# B&R Automation Studio project AriesV2
Automation Studio 4.2.7.54 SP

## Configuration Config_Deployment

### Hardware
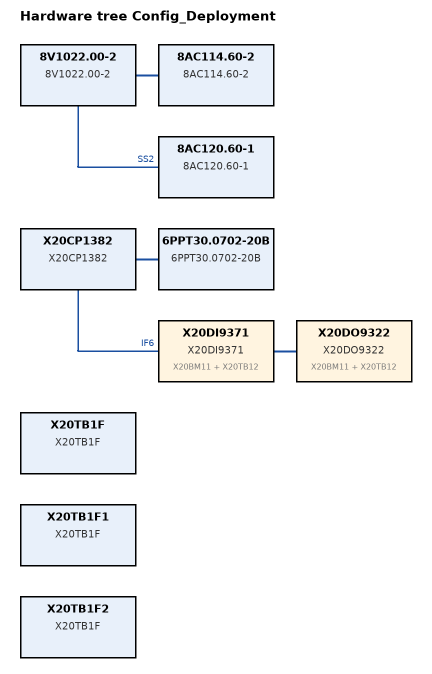
```
6PPT30.0702-20B : 6PPT30.0702-20B v1.1.0.0  [ETH1 -> X20CP1382.IF2 (NodeNumber=1)]
  Terminal = true
  Startmode = 1
  ShowBootlogoVNC = 1
  Mode = Manual
  InternetAddress = 192.168.10.20
  DefaultGateway = 192.168.10.1
  Subnetmask = 255.255.255.0
  Displaybrightness = 75
  SelectedFavoriteVNC = 192.168.10.10
  Favorites_VNC1 = 192.168.10.10
  PasswordVNC = 
  PasswordCIFS = 
  PasswordService = 
  PPTImage = PPT_30_V1.1.1
  VncRefreshRate = 200
8AC114.60-2 : 8AC114.60-2 v1.0.0.8  [SS -> 8V1022.00-2.SS1; PLK1 -> X20CP1382.IF3 (NodeNumber=2)]
8AC120.60-1 : 8AC120.60-1 v1.0.0.2  [SS -> 8V1022.00-2.SS2]
8V1022.00-2 : 8V1022.00-2 v1.0.0.2
  AxisIsPeriodic_r1 = on
  BothEndSwitchesAreNormallyOpen_r1 = on
  QuickStopIsNormallyOpen_r1 = on
X20BM11 : X20BM11 v1.0.0.1  [X2X1 -> X20CP1382.IF6]
X20BM11a : X20BM11 v1.0.0.1  [X2X1 -> X20BM11.X2X2]
X20CP1382 : X20CP1382 v1.3.0.0  [X1 -> X1.SL; X2 -> X2.SL; X3 -> X3.SL]
  Module X1 (Type=X1, Virtual=true, Version=1.0.0.0)
    Connection (Connector=SS1, TargetModule=X20TB1F, TargetConnector=SS)
    Connection (Connector=SL, TargetModule=X20CP1382, TargetConnector=X1)
  Module X2 (Type=X2, Virtual=true, Version=1.0.0.0)
    Connection (Connector=SS1, TargetModule=X20TB1F1, TargetConnector=SS)
    Connection (Connector=SL, TargetModule=X20CP1382, TargetConnector=X2)
  Module X3 (Type=X3, Virtual=true, Version=1.0.0.0)
    Connection (Connector=SS1, TargetModule=X20TB1F2, TargetConnector=SS)
    Connection (Connector=SL, TargetModule=X20CP1382, TargetConnector=X3)
  Connector IF2:
    ActivateDevice = 1
    HostName = x20cpu
    Mode = Manual
    InternetAddress = 192.168.10.10
    SubnetMask = 255.255.255.0
    InaNodeNumber = 0
    Vnc1
    VncVcObjectName1 = Visup
    VncKeyMappingFile1 = VC\PS2-Keyboard4.dis
    VncRefreshRate1 = 200
  Connector IF3:
    CycleTime = 4000
  Connector IF6:
    CycleTime = 4000
  ConfigurationID = AriesV2_Config_Test
  UserPartitionSize = 256
  Simulation = 1
  UserRamSize = 5000
  RemMemSize = 25000
  PermanentPvSize = 15000
  VolatileGlobalPvSize = 300000
  RebootReset = 2
  RebootPowerfail = 2
  TimerDeviceType = EPLX2X
  TimerDevice = X20CP1382.IF3
  TaskClassIdleTime = 8000
  Cyclic1Duration = 4000
  Cyclic1Tolerance = 0
  Cyclic2Duration = 16000
  Cyclic2Tolerance = 16000
  Cyclic3Duration = 48000
  Cyclic3Tolerance = 48000
  Cyclic4Duration = 96000
  Cyclic4Tolerance = 96000
  Cyclic5Duration = 200000
  Cyclic5Tolerance = 200000
  Cyclic6Duration = 496000
  Cyclic6Tolerance = 496000
  Cyclic7Duration = 1000000
  Cyclic7Tolerance = 1000000
  Cyclic8Duration = 8000
  Cyclic8Tolerance = 30000000
  FileDevice1
  FileDeviceName1 = ROOT
  FileDevicePath1 = F:\
  FileDevice2
  FileDeviceName2 = Config
  FileDevicePath2 = F:\Config
  FileDevice3
  FileDeviceName3 = Recipe
  FileDevicePath3 = F:\Recipe
  FileDevice4
  FileDeviceName4 = Process
  FileDevicePath4 = F:\Process
  FtpUser1
  FtpUsername1 = admin
  FtpUserPassword1 = tXcQUdKIsoY/H/jtKSqzHLRzyWbO/eZFb+QmJVs8vuM=
  FtpUserSalt1 = fFlgpUU6
  FTPAccessRight1 = 0
  FTPdevice1 = ALL
  FtpUser2
  FtpUsername2 = user
  FtpUserPassword2 = M/sBBWLbPcMSL0ECBo9+NNWk5QFExAfaSSh+paOlJpQ=
  FtpUserSalt2 = diDYFxUT
  FTPAccessRight2 = 0
  FTPMSpath2 = /
X20DI9371 : X20DI9371 v1.0.1.3  [SS1 -> X20TB12.SS; SL -> X20BM11.SL1]
  Supervision = off
X20DO9322 : X20DO9322 v1.0.3.0  [SS1 -> X20TB12a.SS; SL -> X20BM11a.SL1]
  Supervision = off
X20TB12 : X20TB12 v1.0.0.0
X20TB12a : X20TB12 v1.0.0.0
X20TB1F : X20TB1F v1.0.0.0
X20TB1F1 : X20TB1F v1.0.0.0
X20TB1F2 : X20TB1F v1.0.0.0
```

### Acp10map.ncm - X20CP1382/Motion/Acp10map.ncm
```
NcMapping (NcSwId=Acp10, DisabledNodesAreHidden=False)
  NcObject Axis1 (ModuleId=8V1022.00-2, Type=ncAXIS, Channel=1, AcoposSimulation=Off, InitParameter=Axisi, AcoposParameter=Axisa, AdditionalData=PLCopen_ModPos="1000,1" , Disabled=FALSE, ModuleDisabled=FALSE)
  NcObject 8V1045.00-2_ncV_AXIS1 (ModuleId=8V1022.00-2, Type=ncV_AXIS, Channel=1, Disabled=TRUE, ModuleDisabled=FALSE)
```

### Alarm.mpalarmbasic - X20CP1382/mapp/Alarm.mpalarmbasic
```
Element Alarm_MpLink (Type=mpalarmbasic)
  mapp.Alarm.Factory:
    Reactions:
      Reaction[0]:
        Description = Example: Immediate Stop
  Alarms:
    UserAlarm:
      Alarms:
        Alarm[0]:
          Description = Example: Temperature over Tolerance
          Reaction = 1
```

## Configuration Config_Test

### Hardware
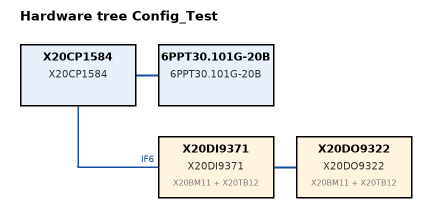
```
6PPT30.101G-20B : 6PPT30.101G-20B v1.1.0.0  [ETH1 -> X20CP1584.IF2 (NodeNumber=1)]
  Terminal = true
  Startmode = 1
  Mode = Manual
  ScreenRotation = 90
  SelectedFavoriteVNC = 192.168.10.10
  PasswordVNC = 
  PasswordCIFS = 
  PasswordService = 
  VncKeyMappingFile = VC\6PPT30.101G-20B.dis
  VncPortNumber = 5901
  VncRefreshRate = 100
  InternetAddress = 192.168.10.20
  DefaultGateway = 192.168.10.1
  Subnetmask = 255.255.255.0
X20BM11 : X20BM11 v1.0.0.1  [X2X1 -> X20CP1584.IF6]
X20BM11a : X20BM11 v1.0.0.1  [X2X1 -> X20BM11.X2X2]
X20CP1584 : X20CP1584 v1.3.2.0
  Connector IF2:
    ActivateDevice = 1
    EthInterfaceRedundant = 0
    HostName = x20cpu
    Mode = Manual
    InternetAddress = 192.168.10.10
    SubnetMask = 255.255.255.0
    Vnc1
    VncVcObjectName1 = Visu1
    VncKeyMappingFile1 = VC\PS2-Keyboard4.dis
    VncRefreshRate1 = 200
  Connector IF3:
    EplInterfaceRedundant = 0
    CycleTime = 8000
    EplEthInterfaceRedundant = 0
  Connector IF6:
    CycleTime = 8000
  ConfigurationID = AriesV2_Config_Test
  UserRamSize = 5000
  RemMemSize = 25000
  PermanentPvSize = 15000
  VolatileGlobalPvSize = 300000
  RebootReset = 2
  RebootPowerfail = 2
  TimerDeviceType = EPLX2X
  TimerDevice = X20CP1584.IF3
  TaskClassIdleTime = 8000
  Cyclic1Duration = 8000
  Cyclic1Tolerance = 0
  Cyclic2Duration = 16000
  Cyclic2Tolerance = 16000
  Cyclic3Duration = 48000
  Cyclic3Tolerance = 48000
  Cyclic4Duration = 96000
  Cyclic4Tolerance = 96000
  Cyclic5Duration = 200000
  Cyclic5Tolerance = 200000
  Cyclic6Duration = 496000
  Cyclic6Tolerance = 496000
  Cyclic7Duration = 1000000
  Cyclic7Tolerance = 1000000
  Cyclic8Duration = 8000
  Cyclic8Tolerance = 30000000
  FileDevice1
  FileDeviceName1 = ROOT
  FileDevicePath1 = F:\
  FileDevice2
  FileDeviceName2 = Config
  FileDevicePath2 = F:\Config
  FileDevice3
  FileDeviceName3 = Recipe
  FileDevicePath3 = F:\Recipe
  FileDevice4
  FileDeviceName4 = Process
  FileDevicePath4 = F:\Process
X20DI9371 : X20DI9371 v1.0.2.0  [SS1 -> X20TB12.SS; SL -> X20BM11.SL1]
  Supervision = off
X20DO9322 : X20DO9322 v1.0.3.0  [SS1 -> X20TB12a.SS; SL -> X20BM11a.SL1]
  Supervision = off
X20TB12 : X20TB12 v1.0.0.0
X20TB12a : X20TB12 v1.0.0.0
```

## Logical view

Binary libraries used (declarations not repeated): operator, runtime, astime, AsIecCon, FileIO, AsXml, standard, brsystem, sys_lib, AsANSL, AsARCfg, AsBrMath, AsBrStr, DataObj, AsTCP, AsUDP, AsUSB, AsArSdm, AsIOTime, AsMem, AsArLog, AsArProf, MTTypes, MTData, wbrListSvc, AsICMP, MpCom, MpAxis, MpWebXs 1.60.1, MpRecipe 1.60.1, MpAlarm, MpFile, Acp10man, Acp10par, NcGlobal, Acp10_MC, Acp10sim, ArTextSys

### BR_AutomationStudio_Winmerge_Settings.txt
```
## This is a directory/file filter for WinMerge
## This filter lets through only files ASP.NET developers care about
name: Exclude Source Control
desc: Exclude Source Control files and directories

## This is an inclusive (loose) filter
## (it lets through everything not specified)
def: include

## Filters for filenames begin with f:
## Filters for directories begin with d:
## (Inline comments begin with " ##" and extend to the end of the line)

## f: \.bzrignore$ ## Bazaar ignore file
## f: \.cvsignore$ ## CVS ignore file
## f: \.gitignore$ ## Git ignore file
## f: \.hgignore$ ## Mercurial ignore file
## f: \.svnignore$ ## Subversion ignore file
## f: \.set$ ## User specific B&R Automation Studio settings
## f: \.state$ ## Even more user specific B&R Automation Studio settings
## f: \.bak$ ## Windows shadow copy files- ignore

f: \.(vs[sp])?scc$  ## Visual SourceSafe files

d: \\\.svn$ ## Subversion working copy
d: \\_svn$  ## Subversion working copy ASP.NET Hack
d: \\cvs$   ## CVS control directory
d: \\\.git$ ## Git directory
d: \\\.bzr$ ## Bazaar branch
d: \\\.hg$ ## Mercurial repository
```

### Global.var
```iecst
VAR CONSTANT
	FORCEIO_ACCESS_LEVEL : UINT := 1;
	CONFIG_ACCESS_LEVEL : UINT := 2;
	RECIPE_ACCESS_LEVEL : UINT := 1;
	DEFINE_MENU_L_HIDE_TIMEOUT_MS : UDINT := 7000;
	DEFINE_MENU_R_HIDE_TIMEOUT_MS : UDINT := 7000;
	DEFINE_HMI_SPLASHSCREEN_TO_MS : UDINT := 5000;
	MAX_IDX_TOTAL_RECIPES : UINT := 100;
	DEFINE_LOGIN_TO : REAL := 600;
END_VAR
(*Insert your comment here.*)
VAR CONSTANT
	MAX_IDX_CREASES : UDINT := 19;
END_VAR
(*Insert your comment here.*)
(*Insert your comment here.*)
VAR RETAIN
	gRecCfg : Global_Par_typ;
END_VAR
VAR
	gAcknowledge : Machine_Alarms_typ;
	gAlarms : Machine_Alarms_typ;
	gMachineName : {REDUND_UNREPLICABLE} STRING[80] := 'Aries';
	gProjectDate : {REDUND_UNREPLICABLE} STRING[80] := '10. April 2017';
	gVersion : {REDUND_UNREPLICABLE} STRING[80] := 'R741';
END_VAR
(*Insert your comment here.*)
VAR
	Axis1 : ACP10AXIS_typ;
	AxisControl : MpAxisBasic;
	AxisPar : MpAxisBasicParType;
	Alarm_Feed : MpAlarmBasicUIConnect20Type := (0);
	Alarm_Feed_UI : MpAlarmBasicUI := (0);
END_VAR
(*Insert your comment here.*)
VAR
	MachineState : AriesMachineState_Enum;
	ProcessState : CreaserPrcsState_Enum;
END_VAR
(*Insert your comment here.*)
VAR
	IO : AriesIOPoints_typ;
	IO_LastCycle : AriesIOPoints_typ;
END_VAR
(*Insert your comment here.*)
VAR
	AppAlarms : MpAlarmBasicUIConnect20Type;
	AppAlarms_FBK : MpAlarmBasic;
	AppAlarms_UI : USINT;
END_VAR
(*Insert your comment here.*)
VAR RETAIN
	gStatistics : Global_Statistics_typ;
END_VAR
(*Insert your comment here.*)
VAR
	gAlarmResetRequested : BOOL;
	StartUIButton_Hide : USINT;
	StopUIButton_Hide : USINT;
	BoardEjectUIButton_Hide : USINT;
	iManualBoardEject : BOOL;
	iMachineErrorReset : BOOL;
	iStartCommand : BOOL;
	iSoftStopCommand : BOOL;
	gSimulateMachine : BOOL;
END_VAR
(*Insert your comment here.*)
VAR CONSTANT
	DEFINE_MM_ROLLER_REV : REAL := 125.664;
END_VAR
VAR
	delta_Board_Position : REAL;
	RollerPos_LastCycle : REAL;
	RollerPos_ThisCycle : REAL;
	Current_Board_Position : REAL;
	Latch_Board_Length : REAL;
	Current_Crease_Section_Length : REAL;
END_VAR
(*Insert your comment here.*)
(*Insert your comment here.*)
```

### Machine.typ
```iecst
TYPE
	CreaserPrcsState_Enum :
		( (*Make sure the indices entered below line up with the VC texts displayed on the UI*)
		PRCS_STATE_INIT := 0,
		PRCS_STATE_READY := 1,
		PRCS_STATE_FEED_BOARD := 2,
		PRCS_STATE_MOVE_CREASE := 3,
		PRCS_STATE_CREASE := 4,
		PRCS_STATE_MOVE_CREASE_WIDTH := 5,
		PRCS_STATE_ERROR := 6,
		PRCS_STATE_EJECT_FINISHED_BOARD := 7,
		PRCS_STATE_SOFT_STOP := 8,
		PRCS_STATE_MOVE_PHOTOEYE_OFFSET := 9
		);
	AriesMachineState_Enum :
		( (*Make sure the indices entered below line up with the VC texts displayed on the UI*)
		MACHINE_STATE_INIT := 0,
		MACHINE_STATE_IDLE := 1,
		MACHINE_STATE_RUNNING := 2,
		MACHINE_STATE_ERROR := 3,
		MACHINE_STATE_HARDWARE_INIT := 4,
		MACHINE_STATE_AXIS_POWER := 5,
		MACHINE_STATE_AXIS_HOME := 6,
		MACHINE_STATE_MANUAL_EJECT := 7
		);
END_TYPE

(*Insert your comment here.*)

TYPE
	CreaserConfig_typ : 	STRUCT
		FeedAxisAccel : REAL;
		FeedAxisDecel : REAL;
		PhotoEyeOffset : REAL;
		PreInsertSpeed : REAL;
		BoardLengthTolerance : REAL;
		CreaseInfeedDelay : REAL;
	END_STRUCT;
	AriesCreaserParams_typ : 	STRUCT
		CreaseDistance_mm : ARRAY[0..MAX_IDX_CREASES]OF REAL;
		CreaseWidth_mm : REAL;
		CreaseCount : UDINT;
		ShaftSensorEdge : UDINT;
		CreaserDirection : UDINT;
		CreaserMotorIdxLag_S : REAL;
		TotalBoardLength : REAL;
	END_STRUCT;
END_TYPE

(*Insert your comment here.*)

TYPE
	AriesIOPoints_typ : 	STRUCT
		oCreaserCCWRotation : BOOL;
		oCreaserCWRotation : BOOL;
		oBoardFeedingLight : BOOL;
		oUIIndicatorLight : BOOL;
		iSafeMachineState : BOOL;
		iCreaserShaftSensor : BOOL;
		iFiberOpticSensor : BOOL;
		iSM1Disabled : BOOL;
	END_STRUCT;
END_TYPE

(*Insert your comment here.*)

TYPE
	Machine_Alarms_typ : 	STRUCT  (*Did something fancy here- structure is copied into array for VC error texts, make sure the following numbers line up with the VC error text indices!*)
		SM1_Disabled : BOOL; (*0*)
		Unsafe_Machine_State : BOOL; (*1*)
		Fiber_Optic_Blocked_RunCmd : BOOL; (*2*)
		Creaser_Shaft_Edge_Timeout : BOOL; (*3*)
		Error_State_Unsafe_Machine : BOOL; (*4*)
		Error_State_SM1_Power : BOOL; (*5*)
		Feed_Axis_Motor_Error : BOOL; (*6*)
		Crease_Count_Greater_Max : BOOL; (*7*)
		Error_State_Process_Error : BOOL; (*8*)
		Load_Recipe : BOOL; (*9*)
		Manual_Home_Creaser_Blade : BOOL; (*10*)
		Board_Length_GT_Confgd_Amount : BOOL; (*11*)
		Board_Length_LT_Confgd_Amount : BOOL; (*12*)
		Measured_Length_GT_Configured : BOOL; (*13*)
		Measured_Length_LT_Configured : BOOL; (*14*)
		Unsaved_Recipe_Params : BOOL; (*15*)
	END_STRUCT;
	Global_Statistics_typ : 	STRUCT
		total_runtime : UDINT;
		runtime_h : UDINT;
		runtime_m : UDINT;
		runtime_s : UDINT;
		total_processed : UDINT;
		Reset : BOOL;
		total_creases : UDINT;
		Sum_Board_Travel_Lengths : REAL;
		Avg_Board_Length : REAL;
	END_STRUCT;
END_TYPE
```

### Generic_Rec_Cfg.typ
```iecst
TYPE
	HMIConfig_typ : 	STRUCT
		passwordSetup : STRING[15];
		passwordEngineer : STRING[15];
		passwordFactory : STRING[15];
		MachineLang : UDINT;
	END_STRUCT;
END_TYPE

(*Insert your comment here.*)

TYPE
	Global_Rec_typ : 	STRUCT
		MagicPrefix : UDINT;
		FeedVelocity : REAL;
		Crease : AriesCreaserParams_typ;
		MagicSuffix : UDINT;
	END_STRUCT;
	Global_Cfg_typ : 	STRUCT
		MagicPrefix : UDINT;
		Creaser : CreaserConfig_typ;
		HMI : HMIConfig_typ;
		wbrMemService : wbrMemService_typ;
		cfgCompile : cfgCompileVersionInfo_typ;
		MagicSuffix : UDINT;
	END_STRUCT;
END_TYPE

(*Insert your comment here.*)

TYPE
	Global_Rec_Cfg_typ : 	STRUCT
		Rec : Global_Rec_typ;
		Cfg : Global_Cfg_typ;
	END_STRUCT;
	Global_RecCfg_Public_In_typ : 	STRUCT
		Copy_default_to_save : USINT;
		Copy_default_to_active : USINT;
		Copy_save_to_active : USINT;
		Copy_save_to_default : USINT;
		Copy_active_to_save : USINT;
		Copy_active_to_default : USINT;
		Copy_internal_to_default : USINT;
		FileName : STRING[255];
	END_STRUCT;
	Global_RecCfg_Public_Out_typ : 	STRUCT
		save_differs_from_active : USINT;
		default_differs_from_save : USINT;
		active_differs_from_default : USINT;
		Initial_Load : USINT;
	END_STRUCT;
	Global_Rec_Cfg_Info_typ : 	STRUCT
		O : Global_RecCfg_Public_Out_typ;
		I : Global_RecCfg_Public_In_typ;
	END_STRUCT;
	Global_Rec_Cfg_IO_typ : 	STRUCT
		Rec : Global_Rec_Cfg_Info_typ;
		Cfg : Global_Rec_Cfg_Info_typ;
	END_STRUCT;
	Global_Par_typ : 	STRUCT
		save : Global_Rec_Cfg_typ;
		active : Global_Rec_Cfg_typ;
		defaultvals : Global_Rec_Cfg_typ;
		IO : Global_Rec_Cfg_IO_typ;
	END_STRUCT;
END_TYPE

(*Insert your comment here.*)
```

### Package Logical/Libraries - Global libraries

### Library Logical/Libraries/jgLibC (ANSIC)
Depends on: standard

#### Indexer_Helper_functions.c
```c
/********************************************************************
 * COPYRIGHT -- Microsoft
 ********************************************************************
 * Library: jgLibC
 * File: Indexer_Helper_functions.c
 * Author: Admin
 * Created: May 11, 2015
 *******************************************************************/

#include <bur/plctypes.h>
#include <jgLibC.h>
UDINT Tms(REAL in){
	UDINT var_return = 0;

	var_return = (UDINT) (1000 * in);

	return var_return;
}
```

### Library Logical/Libraries/MAPPSuppor (ANSIC) - library (written/managed by J. Glisson) containing functions for ACPu err acknowledgement, HMI param table construction, HMI param table activation to the common layer

#### HMIparamList.typ
```iecst
(********************************************************************
 * COPYRIGHT -- piedmont
 ********************************************************************
 * Package: HMI
 * File: HMI.typ
 * Author: goran
 * Created: August 28, 2013
 ********************************************************************
 * Data types of package HMI
 ********************************************************************)
(*########################################################################*)
(*HMI object - PARAMETER LIST - LIMITS*)
(*########################################################################*)
(*########################################################################*)
(*HMI object - PARAMETER LIST*)
(*########################################################################*)

TYPE
	HMITableIndex_enum :
		(
		TABLE_RECIPE := 0,
		TABLE_CONFIG := 1
		);
	hmiTableStatStruct_typ : 	STRUCT
		maxLenDesc : UDINT;
		maxLenName : UDINT;
		Param : UDINT;
		Default : UDINT;
		Min : UDINT;
		Max : UDINT;
		Hide : UDINT;
	END_STRUCT;
	hmiTableStats_typ : 	STRUCT
		Overall : hmiTableStatStruct_typ;
	END_STRUCT;
	PVList_Language_Texts_typ : 	STRUCT
		PVTextLangSpecific : STRING[DEFINE_PAR_NAME_MAXLEN];
		PVDescLangSpecific : STRING[DEFINE_PAR_DESC_MAXLEN];
	END_STRUCT;
	PVListTexts_Info_typ : 	STRUCT
		Str : STRING[DEFINE_PAR_NAME_MAXLEN];
		isValid : BOOL;
		isPV : BOOL;
		isConstant : BOOL;
		Const_Value : REAL;
		PVAdr : {REDUND_UNREPLICABLE} UDINT;
		PVLen : USINT;
		PVDim : USINT;
		PVTyp : UDINT;
		StrLen : UDINT;
	END_STRUCT;
	PVTable_Val_Info_typ : 	STRUCT
		Param : PVListTexts_Info_typ;
		Default : PVListTexts_Info_typ;
		Min : PVListTexts_Info_typ;
		Max : PVListTexts_Info_typ;
		Hide : PVListTexts_Info_typ;
	END_STRUCT;
	PVTableInfo : 	STRUCT
		PVText : ARRAY[0..MAX_IDX_LANGUAGES]OF PVList_Language_Texts_typ;
		Val : PVTable_Val_Info_typ;
		Error : BOOL;
	END_STRUCT;
	HMI_Table_Data_typ : 	STRUCT
		info : ARRAY[0..DEFINE_MAX_TABLE_ENTRIES]OF PVTableInfo;
		Max_Idx_Entries : UDINT;
		Table_Name : STRING[DEFINE_PAR_NAME_MAXLEN];
		NameSpace : STRING[DEFINE_PAR_NAME_MAXLEN];
		Load_OK : BOOL;
	END_STRUCT;
	hmiParamLimits_typ : 	STRUCT
		k_factor : REAL; (*scaling k factor (y=kx + n, where y=dsiplay value, x=plc value)*)
		n_factor : REAL; (*scaling n factor (y=kx + n, where y=dsiplay value, x=plc value)*)
		minValue : REAL; (*min value*)
		maxValue : REAL; (*max value*)
		defaultValue : REAL; (*default value*)
		pEnumText : UDINT; (*ptr to a string of comma delimited enum texts*)
		pEnumVals : UDINT; (*ptr to a string of comma delimited enum values*)
		valueType : UINT; (*type of the paramvalue (0-DINT, 1-REAL, 2-ENUM)*)
	END_STRUCT;
	hmiParamListTable_typ : 	STRUCT
		listHeader : STRING[DEFINE_PAR_NAME_MAXLEN]; (*name of the list (header text)*)
		listIdText : ARRAY[0..DEFINE_MAX_TABLE_ENTRIES]OF STRING[DEFINE_PAR_IDX_MAXLEN]; (*table colum: id-s*)
		listTypeText : ARRAY[0..DEFINE_MAX_TABLE_ENTRIES]OF STRING[DEFINE_PAR_NAME_MAXLEN]; (*table colum: value*)
		listDefaultText : ARRAY[0..DEFINE_MAX_TABLE_ENTRIES]OF STRING[DEFINE_PAR_NAME_MAXLEN]; (*table colum: value*)
		listMinText : ARRAY[0..DEFINE_MAX_TABLE_ENTRIES]OF STRING[DEFINE_PAR_NAME_MAXLEN]; (*table colum: value*)
		listMaxText : ARRAY[0..DEFINE_MAX_TABLE_ENTRIES]OF STRING[DEFINE_PAR_NAME_MAXLEN]; (*table colum: value*)
		listValueText : ARRAY[0..DEFINE_MAX_TABLE_ENTRIES]OF STRING[DEFINE_PAR_NAME_MAXLEN]; (*table colum: value*)
		listName : ARRAY[0..DEFINE_MAX_TABLE_ENTRIES]OF STRING[DEFINE_PAR_NAME_MAXLEN]; (*table colum: name*)
		listDescription : ARRAY[0..DEFINE_MAX_TABLE_ENTRIES]OF STRING[DEFINE_PAR_DESC_MAXLEN]; (*table colum: description*)
		listValuePtr : ARRAY[0..DEFINE_MAX_TABLE_ENTRIES]OF UDINT; (*list of ptrs to parametars*)
		listDecPlaces : ARRAY[0..DEFINE_MAX_TABLE_ENTRIES]OF DINT; (*list of dec places for each parametar*)
		listLimits : ARRAY[0..DEFINE_MAX_TABLE_ENTRIES]OF hmiParamLimits_typ;
		selName : {REDUND_UNREPLICABLE} STRING[DEFINE_PAR_NAME_MAXLEN]; (*name of the currently selected/active parametar*)
		selDescription : STRING[DEFINE_PAR_DESC_MAXLEN]; (*description of the currently selected/active parametar*)
		selValueEnumIndex : UDINT; (*value of the currently selected/active parametar for type enum*)
		selValueEnumIndexMax : UDINT; (*value of the currently selected/active parametar for type enum*)
		selValueREAL : REAL; (*value of the currently selected/active parametar*)
		selValueREALOld : REAL; (*value of the currently selected/active parametar (previous value for change detection*)
		selValueREALMax : REAL; (*max value of the currently selected/active parametar*)
		selValueREALMin : REAL; (*min value of the currently selected/active parametar*)
		selValueREALDefault : REAL; (*default value of the currently selected/active parametar*)
		selValueDecPlaces : DINT; (*default value of the currently selected/active parametar*)
		selValueDINT : DINT; (*value of the currently selected/active parametar*)
		selValueDINTOld : DINT; (*value of the currently selected/active parametar (previous value for change detection*)
		selValueDINTMax : DINT; (*max value of the currently selected/active parametar*)
		selValueDINTMin : DINT; (*min value of the currently selected/active parametar*)
		selValueDINTDefault : DINT; (*default value of the currently selected/active parametar*)
		selValueFormVisible : DINT; (*visibility control of the form / controls for setting parametar value*)
		index : UINT; (*index of the currently selected/active parametar*)
		indexOld : UINT; (*index of the currently selected/active parametar (previous value for change detection)*)
		maxIndex : UINT; (*max index / number of items in the table. Must be less then hmiTableMAXDESCRIPTION!!!*)
		setDefaultRequest : BOOL; (*set default request flag*)
		incDP : USINT;
		decDP : USINT;
	END_STRUCT;
END_TYPE
```

#### hmiParamList.h
```c
/********************************************************************
 * COPYRIGHT -- piedmont
 ********************************************************************
 * Program: hmilogic
 * File: hmiParamList.h
 * Author: goran
 * Created: September 05, 2013
 *******************************************************************/
#include <bur/plctypes.h>
#ifdef _DEFAULT_INCLUDES
#include <AsDefault.h>
#endif
//void hmiParamListTableCyclic(hmiParamListTable_typ* p);
void hmiParamListTableEntryLast(hmiParamListTable_typ* p);
void hmiParamListTableEntryFirst(hmiParamListTable_typ* p, char* pListName);
 void hmiParamListTableAddEntryNext(hmiParamListTable_typ* p, UDINT pValue, char* pName, REAL valDefault, REAL valMin, REAL valMax, DINT decPlaces, REAL k_factor, REAL n_factor, UINT valueType, char* pDescription);
```

#### hmiParamList.c
```c
/********************************************************************
 * COPYRIGHT -- piedmont
 ********************************************************************
 * Program: hmilogic
 * File: hmiParamList.c
 * Author: goran
 * Created: September 05, 2013
 *******************************************************************/

#include <bur/plctypes.h>
#ifdef _DEFAULT_INCLUDES
	#include <AsDefault.h>
#endif

#include <AsBrStr.h>

#define HMI_PARAMLIST_DECPLACES_DEFAULT  2 //default value of decimal places for any real number converted to text. Application specific.

/*
###############################################################################
HMI table editor support. Set of functions that support table based editing of the parametars.
###############################################################################
*/

/**
rouding of a floating point value to the number of required decimal positions.
\param d value
\param pp number of decimal places
\return rounded value

*/
static float roundVal(float d, int ppOffset)
{

	int valInt;
	float exp10topp = 10.0;
	int count = 0;
	int pp = ppOffset;

	if(!pp){
		exp10topp = 1.0;
	}else
		if(pp<0){
		exp10topp = 0.1;
		count = (0 - pp) - 1;
	}else{
		exp10topp = 10.0;
		count = pp - 1;
	}

	while(count--){
		exp10topp *= exp10topp;
	}

	valInt = (int) (d *  exp10topp + 0.5);
	return ( valInt  /  exp10topp  );
}

/**
ftoa (float to ascii converion) with the added support for required number of decimal places in the text ouput.
\param value value to convert
\param pp number of decimal places
\return rounded value

*/
static void ftoaEx(float value, char* pText, int decPlacesOffset)
{
	char text[32];

	int len;
	int comaPos;
	int apendZerosCount;
	int ii;
	float rnd_val;
	int decPlaces = HMI_PARAMLIST_DECPLACES_DEFAULT + decPlacesOffset;

	if(!pText)
		return;

	//limit max dec places
	if(decPlaces > 5)
		decPlaces = 5;

	//convert float to ascii
	//	ftoa(value, text);
	rnd_val = roundVal(value, decPlaces);
	brsftoa(rnd_val , (UDINT)text);

	//get the length of the converted string
	len = strlen(text);
	if(!len){
		//0 length > don't know what to do
		strcpy(pText, "?");
		return;
	}

	//find position of the coma
	comaPos = bgStrFind(text, ".", -1, -1);

	if(!decPlaces){
		//dec places are not needed

		if(comaPos>0){
			//coma is present > terminate the string at the comma position
			text[comaPos] = 0;
		}

	}else{
		//dec places are needed

		if(comaPos<0){
			//no coma present but it is needed
			strcat(text, ".");
			len+=1;
			comaPos=len-1;
		}

		apendZerosCount = decPlaces - (len - comaPos - 1);

		if(apendZerosCount < 0){
			//too many digits after a decimal place > terminate string to a specified number of dec places
			apendZerosCount = 0 - apendZerosCount;
			text[len - apendZerosCount]=0;
		}else{
			//need to add zeros to satisfy the number of dec places
			for(ii=0; ii<apendZerosCount; ii++){
				text[len+ii]='0';
			}
			text[len+ii]=0;
		}
	}

	strcpy(pText, text);
	return;
}

static float hmiParamListTableGetPLCValue(UDINT pValue, REAL k_factor, REAL n_factor, int valueType)
{
	UDINT* pUdint = (UDINT*)pValue;
	float* pFloat = (float*)pValue;
	REAL tempReal;

	switch(valueType){
		case 1:
			if(pFloat){
				tempReal = ((float)(*pFloat)) * k_factor + n_factor;
			}else{
				tempReal = 0.0;
			}
			break;
		default:
			if(pUdint){
				tempReal = ((float)(*pUdint)) * k_factor + n_factor;
			}else{
				tempReal = 0.0;
			}
			break;
	}

	return tempReal;
}

static void hmiParamListTableDisplayToValue(float value, UDINT pValue, char* pOutputText,  int decPlaces, REAL k_factor, REAL n_factor, int valueType)
{
/*
scaling
y=kx + n
y=display value
x=plc value

x = (y- n)*(1/k)

value types:
0-UDINT
1-REAL

*/

	UDINT* pUdint = (UDINT*)pValue;
	float *pFloat = (float*)pValue;

	if(!k_factor){
		strcpy(pOutputText, "ERR: div by 0");
		return;
	}

	switch(valueType){
		case 1:
			*pFloat = (float)((value - n_factor) / k_factor);
			break;
		default:
			*pUdint = (UDINT)((value - n_factor) / k_factor);
			break;
	}

	ftoaEx(value, pOutputText, decPlaces);
}

static void hmiParamListTableValueToDisplay(UDINT pValue, char* pOutputText, float* pOutputFloat, int decPlaces, REAL k_factor, REAL n_factor, int valueType)
{
/*
scaling
y=kx + n
y=display value
x=plc value
*/
	REAL tempReal = hmiParamListTableGetPLCValue(pValue, k_factor, n_factor, valueType);

	if(pOutputFloat)
		*pOutputFloat = tempReal;

	ftoaEx(tempReal, pOutputText, decPlaces);
}

 void hmiParamListTableAddEntryNext(hmiParamListTable_typ* p, UDINT pValue, char* pName,
REAL valDefault, REAL valMin, REAL valMax, DINT decPlaces, REAL k_factor, REAL n_factor, UINT valueType, char* pDescription)
{
	if(p->index >= DEFINE_MAX_TABLE_ENTRIES){
		strcpy(p->listValueText[p->index], "table overflow!");
		return;
	}

	p->listValuePtr[p->index] = pValue;
	bgsprintf(p->listIdText[p->index], "%d", p->index);
	bgStrCpyN(p->listDescription[p->index], pDescription, sizeof(p->listDescription[0]));
	bgStrCpyN(p->listName[p->index], pName, sizeof(p->listName[0]));
	p->listDecPlaces[p->index] = decPlaces;

	switch(valueType){
		case 0:
			bgsprintf(p->listTypeText[p->index], "%s", "INT");
			break;
		case 1:
			bgsprintf(p->listTypeText[p->index], "%s", "FLOAT");
			break;
		default:
			bgsprintf(p->listTypeText[p->index], "%s", "ERR");
			break;
	}

	brsftoa(valDefault,(UDINT) &p->listDefaultText[p->index]);
	brsftoa(valMin,(UDINT) &p->listMinText[p->index]);
	brsftoa(valMax,(UDINT) &p->listMaxText[p->index]);

	p->listLimits[p->index].defaultValue = valDefault;
	p->listLimits[p->index].minValue= valMin;
	p->listLimits[p->index].maxValue= valMax;
	p->listLimits[p->index].k_factor= k_factor;
	p->listLimits[p->index].n_factor= n_factor;
	p->listLimits[p->index].valueType= valueType;

	hmiParamListTableValueToDisplay(p->listValuePtr[p->index],
		p->listValueText[p->index], 0, p->listDecPlaces[p->index], p->listLimits[p->index].k_factor, p->listLimits[p->index].n_factor, p->listLimits[p->index].valueType);

	p->index++;
	p->maxIndex++;
}

void hmiParamListTableEntryFirst(hmiParamListTable_typ* p, char* pListName)
{
	brsmemset((UDINT) p, 0, sizeof(hmiParamListTable_typ));
	p->maxIndex = 0;
	p->index = 0;
	bgStrCpyN(p->listHeader, pListName, sizeof(p->listHeader));
}

void hmiParamListTableEntryLast(hmiParamListTable_typ* p)
{
	if(p->maxIndex)
		p->maxIndex--;

	//init index value
	p->index = 0;

	//update text fields according to the currently selected table element
	bgStrCpyN(p->selName, p->listName[p->index], sizeof(p->selName));
	bgStrCpyN(p->selDescription, p->listDescription[p->index], sizeof(p->selDescription));

	//set limits on the HMI input control that coresponds to the currently selected table element
	p->selValueREALMin = p->listLimits[p->index].minValue;
	p->selValueREALMax= p->listLimits[p->index].maxValue;
	p->selValueREALDefault = p->listLimits[p->index].defaultValue;
	p->selValueDecPlaces = p->listDecPlaces[p->index];

	//display selected table element
	hmiParamListTableValueToDisplay(p->listValuePtr[p->index],
		p->listValueText[p->index], &p->selValueREAL, p->listDecPlaces[p->index], p->listLimits[p->index].k_factor, p->listLimits[p->index].n_factor, p->listLimits[p->index].valueType);

}

USINT hmiParamListTableCyclic(UDINT p_int)
{
	hmiParamListTable_typ* p = p_int;

	//limit index to max index value (up arrow)
	if(p->index >= p->maxIndex){
		p->index = p->maxIndex;
	}

	//keep checking if index changes (i.e. user changes entry selection)
	if(p->index != p->indexOld){
		//index change > update selected value for user entry
		p->indexOld = p->index;
		hmiParamListTableValueToDisplay(p->listValuePtr[p->index], p->listValueText[p->index],
			&p->selValueREAL, p->listDecPlaces[p->index], p->listLimits[p->index].k_factor, p->listLimits[p->index].n_factor, p->listLimits[p->index].valueType);
		//store value for change detection
		p->selValueREALOld = p->selValueREAL;

		//update text fields
		bgStrCpyN(p->selName, p->listName[p->index], sizeof(p->selName));
		bgStrCpyN(p->selDescription, p->listDescription[p->index], sizeof(p->selDescription));

		//set limits for the selected element
		p->selValueREALMin = p->listLimits[p->index].minValue;
		p->selValueREALMax= p->listLimits[p->index].maxValue;
		p->selValueREALDefault = p->listLimits[p->index].defaultValue;
		p->selValueDecPlaces = p->listDecPlaces[p->index];

	}

	//keep checking if currently selected value changes(i.e. user enteres new value)
	if(p->selValueREALOld != p->selValueREAL){
		if(p->selValueREALMin < p->selValueREALMax){
			//enforce limits
			if(p->selValueREAL < p->selValueREALMin)
				p->selValueREAL = p->selValueREALMin;

			if(p->selValueREAL > p->selValueREALMax)
				p->selValueREAL = p->selValueREALMax;
		}
		p->selValueREALOld = p->selValueREAL;
		hmiParamListTableDisplayToValue(p->selValueREAL, p->listValuePtr[p->index], p->listValueText[p->index],
			p->listDecPlaces[p->index], p->listLimits[p->index].k_factor, p->listLimits[p->index].n_factor, p->listLimits[p->index].valueType);
	}

	//keep checking if the source of the currently selected value changes on a PLC(i.e. PLC location gets updated, etc)
	{
		float tempVal = hmiParamListTableGetPLCValue(p->listValuePtr[p->index], p->listLimits[p->index].k_factor, p->listLimits[p->index].n_factor, p->listLimits[p->index].valueType);
		if(p->selValueREAL != tempVal){
			//PLC value changed > update displayed value
			p->selValueREAL = tempVal;
			p->selValueREALOld = p->selValueREAL;
			hmiParamListTableDisplayToValue(p->selValueREAL, p->listValuePtr[p->index], p->listValueText[p->index],
				p->listDecPlaces[p->index], p->listLimits[p->index].k_factor, p->listLimits[p->index].n_factor, p->listLimits[p->index].valueType);

		}
	}

	//set default value request?
	if(p->setDefaultRequest){
		p->setDefaultRequest = 0;
		p->selValueREAL = p->selValueREALDefault;
	}
	return 0;
}

//eof
```

### Package Logical/Libraries/wbrServices - Service libraries

### wbrServices.typ
```iecst
(*** /*****************************************************************
 * \copyright -- Piedmont Automation
 ********************************************************************
 * Program : wbrServices
 * \file :   wbrServices.typ
 * \author : Blanton Radford
 * \date Created: July 17, 2015
 ********************************************************************
 * Data types of package wbrServices
 ***************************************************************/ *****)

TYPE
	wbrSvcBool_enum :
		(
		NO := 0,
		YES,
		OFF := 0,
		ON,
		STOP := 0,
		START,
		UNCHECK := 0,
		CHECK
		);
	cfgFileInfo_typ : 	STRUCT
		timestamp : STRING[63];
		path : STRING[127];
		machineNumber : UDINT;
		machineName : STRING[31];
	END_STRUCT;
END_TYPE
```

### wbrServicesGlobal.var
```iecst
(********************************************************************
 * COPYRIGHT -- Piedmont Automation
 ********************************************************************
 * Package: listServices
 * File: listServicesGlobal.var
 * Author: Blanton Radford
 * Created: August 11, 2014
 ********************************************************************
 * Variables of package listServices
 ********************************************************************)
VAR
	memService : wbrMemService_typ := (0);
	logService : wbrLogService_typ := (0);
	genericPing : wbrPingService_typ;
END_VAR
```

### Program Logical/Libraries/wbrServices/bglibasWBR

#### bgfifo.c
```c
/********************************************************************
 * COPYRIGHT -- HP
 ********************************************************************
 * Library: bglibas
 * File: bgfifo.c
 * Author: goran
 * Created: February 01, 2013
 *******************************************************************/

#include <bur/plctypes.h>
#ifdef __cplusplus
	extern "C"
	{
#endif

#include "bglibasWBR.h"

#ifdef __cplusplus
	};
#endif
#include <string.h>

static void bgFIFOPushEntry(bgFIFO_typ* p)
{
	char *pSrc = (char*)p->iPtrPushData;//src data
	char* pDst = (char*)((char*)p->prvFIFOMemory + (p->cfgEntrySize * p->oPushIdx));//empty FIFO location
	memcpy(pDst, pSrc, p->cfgEntrySize);

	p->oPushIdx++;//inc location index to next empty FIFO spot
	if(p->oPushIdx >= p->cfgMaxEntries){
		p->oPushIdx = 0;//handle roll over (ring buffer)
	}

	p->oFIFOCount++;//inc number of FIFO entries
	if(p->oFIFOCount >= p->cfgMaxEntries){
		p->oFIFOFull = 1;//set FIFO full indication
	}
}

static void bgFIFOPullEntry(bgFIFO_typ* p)
{
	char* pSrc = (char*)((char*)p->prvFIFOMemory + (p->cfgEntrySize * p->oPullIdx));//oldest FIFO entry
	char *pDst = (char*)p->oPtrPullData;//destination
	memcpy(pDst, pSrc, p->cfgEntrySize);

	p->oPullIdx++;//inc oldest stored FIFO entry position
	if(p->oPullIdx >= p->cfgMaxEntries){
		p->oPullIdx = 0;//handle roll over (ring buffer)
	}

	if(p->oFIFOCount)//dec number of entris in the FIFO
		p->oFIFOCount--;

	p->oFIFOFull = 0;//reset FIFO full indication
}

/**
bgFIFOInit()
-simple FIFO. Stores upto (entryTotalCount) number of elements. Elements MUST be of the same size.
-supports push/pull action
-push:
- user supplied data is copied into the available FIFO memory space, number of items in the FIFO gets incremented,
index variable that keeps track of next empty FIFO location is adjusted; if FIFO full - no action, error returned
-pull:
- oldest entry from FIFO copied to user supplied data space; number of items in the FIFO gets decremented,
index variable that keeps track of oldeset FIFO entry is adjusted; if FIFO empty - no action, error is returned
*/
unsigned long bgFIFOInit(struct bgFIFO_typ* p, unsigned long  entrySize, unsigned long  entryTotalCount, unsigned long  pFIFOMem)
{
	if(!p || !pFIFOMem || !entrySize || (entryTotalCount <=5))
		return 1;

	p->iPtrPushData = 0;
	p->oPtrPullData = 0;

	p->oFIFOCount = 0;
	p->oFIFOFull = 0;

	p->cfgEntrySize = entrySize;
	p->cfgMaxEntries = entryTotalCount;
	p->prvFIFOMemory = pFIFOMem;
	p->oPullIdx = 0;
	p->oPushIdx = 0;
	return 0;
}

/* Push data to FIFO. Content from pSrc is copied into the available FIFO memory. In case of error return value is != 0*/
unsigned long bgFIFOPush(struct bgFIFO_typ* p, unsigned long pSrc, unsigned long srcSize)
{
	if(!p)
		return 1;

	if(!p->prvFIFOMemory)
		return 2;

	if(!pSrc)
		return 3;

	if(!srcSize || (srcSize != p->cfgEntrySize) )
		return 4;

	if(p->oFIFOFull)
		return 5;

	p->iPtrPushData = pSrc;
	bgFIFOPushEntry(p);
	return 0;
}

/* Pull (retrive) data from FIFO. Oldest entry from FIFO memory is copied into the provided pDst space. In case of error return value is != 0*/
unsigned long bgFIFOPull(struct bgFIFO_typ* p, unsigned long pDst, unsigned long dstSize)
{
	if(!p)
		return 1;

	if(!p->prvFIFOMemory)
		return 2;

	if(!pDst)
		return 3;

	if(!dstSize || (dstSize != p->cfgEntrySize) )
		return 4;

	if(!p->oFIFOCount)
		return 5;

	p->oPtrPullData = pDst;
	bgFIFOPullEntry(p);
	return 0;
}

/* Get the number of entries stored in the FIFO.*/
unsigned long bgFIFOGetCount(struct bgFIFO_typ* p)
{
	if(!p)
		return 0;

	return p->oFIFOCount;
}

/* Check if FIFO is full.*/
unsigned long bgFIFOIsFull(struct bgFIFO_typ* p)
{
	if(!p)
		return 0;

	return p->oFIFOFull;
}
//EOF
```

#### bgTimer1ms.c
```c
/********************************************************************
 * COPYRIGHT -- belgor
 ********************************************************************
 * Package: bglib
 * File: bgTimer1ms.c
 * Author: goran
 * Created: October 05, 2011
 *******************************************************************/
#include <bur/plctypes.h>
#ifdef __cplusplus
	extern "C"
	{
#endif

#include "bglibasWBR.h"

#ifdef __cplusplus
	};
#endif
#include <standard.h>

/* Timer cyclic function. Must be called cyclicly for corret timer operation. */
unsigned long  bgTimerCyclic(struct TON *timer){
	TON(timer);
	return 0;
}

unsigned long  bgTimerOffCyclic(struct TOF *timer){
	TOF(timer);
	return 0;
}

/* Start timer for a defined amount of time [ms]. IMPORTANT: function uses TON library call. Same restrictions apply! */
unsigned long  bgTimerStart(struct TON *timer, unsigned long timeoutTime){
	timer->IN = 0;
	TON(timer);
	timer->IN = 1;
	timer->PT = timeoutTime;
	TON(timer );
	return 0;
}

/* Stop the timer.*/
unsigned long  bgTimerStop(struct TON *timer){
	timer->IN = 0;
	TON(timer);
	return 0;
}

/* Check if timer has expired.*/
BOOL  bgTimerIsTimeOut(struct TON *timer){
	if( bgTimerIsEnabled(timer) ){
		return (timer->Q);
	}else{
		return (1);
	}
}

/* Check if timer is enabled.*/
BOOL  bgTimerIsEnabled(struct TON *timer){
	return (timer->IN);
}

/* Retrive the remainig timer time [ms].*/
unsigned long  bgTimerTimeRemaining(struct TON *timer){
	return (timer->PT - timer->ET);
}

/* Retrive the elapsed timer time [ms].*/
unsigned long  bgTimerTimeElapsed(struct TON *timer) {
	return (timer->ET);
}

//EOF
```

### Program Logical/Libraries/wbrServices/Cyclic/wbrService

#### wbrServiceCyclic.c
```c
/********************************************************************
 * \copyright -- Piedmont Automation
 ********************************************************************
 * Program : wbrService
 * \file :   wbrServiceCyclic.c
 * \author : Blanton Radford
 * \date Created: May 18, 2015
 ********************************************************************
 * \brief Implementation of program wbrService
 ********************************************************************/

#ifdef _DEFAULT_INCLUDES
  #include <AsDefault.h>
#endif

/*! \brief Cyclic task for ?
*   \pre   Place in TC#?
*/
void _CYCLIC wbrServiceCyclic(void)
{
  //! \todo   check available mem and set flags to increase partition size if needed
  memService.status.blockFree=  memSvcGetMemInfo();

  if(logService.busy)  writeMessagesToLog();

  wbrPingStation(&genericPing);
}

void _EXIT wbrServiceExit(void)
{
  if(logService.busy)  writeMessagesToLog();
}
```

### changeLog.txt
```
0.10.7  2016-04
  Clean up some /todos and other comments
  Added wbrMemService to wrap AsMem and allow services besides list service
    to use heap memory
    moved mem funcs and data from wbrListService to wbrMemService

0.10.6  2016-03-31
  Added TimerServices
    Made a few mods to suit Hailo project and be more generic, e.g. msTimer object declared
    Using clock_ms() from AsTime to count milliseconds
    Added msTimer.diff_ms to facilitate time tracking, e.g. "hour meters"
  A few changes to Init and Cyclic to be more generic for multiple projects
    Write compile info to log on Init
  Updated package dependencies to facilitate more trouble-free importing

0.10.5  2015-10-??
  Initial release
    Used in APDW project
    No complaints as of 2016-03-07
```

### TimerServices.var - Package variables
```iecst
(********************************************************************
 * COPYRIGHT -- Piedmont Automation
 ********************************************************************
 * Package: TimerServices
 * File: TimerServices.var
 * Author: Blanton Radford
 * Created: December 05, 2014
 ********************************************************************
 * Variables of package TimerServices
 ********************************************************************)
VAR
	msTimer : msTimer_typ;
END_VAR
```

- Program Logical/Libraries/wbrServices/TimerServices/msTimeSvc (ANSIC) - ms-based time service (no source held here)

### wbrLogSvc.typ
```iecst
(*** /*****************************************************************
 * \copyright -- Piedmont Automation
 ********************************************************************
 * Program : wbrLogSvc
 * \file :   wbrLogSvc.typ
 * \author : Blanton Radford
 * \date Created: May 07, 2015
 ********************************************************************
 * Data types of library wbrLogSvc
 ****************************************************************/ ****)

TYPE
	wbrLogServiceTextLog_typ : 	STRUCT
		view : ARRAY[0..127]OF STRING[127]; (*View window into the log*)
		str : wbrListSvcStringList_typ;
	END_STRUCT;
	wbrLogServiceLogListNode_typ : 	STRUCT
		fb : AsArLogWrite;
		inMsg : STRING[127];
	END_STRUCT;
	wbrLogService_typ : 	STRUCT
		list : linkedList_typ;
		message : STRING[127] := 'no message to output';
		log : wbrLogServiceTextLog_typ;
		logLevel : USINT := 4; (*The higher the value, the more messages are logged, i.e. the log will contain more detail and will grow larger more quickly*)
		busy : BOOL;
		maxNodesUsed : UDINT;
	END_STRUCT;
	wbrLogServiceLogbookInfo_typ : 	STRUCT
		name : STRING[15];
		length : UDINT := 65535;
		memType : UDINT := 2;
		status : UINT;
		ident : UDINT;
		index : UDINT;
		formatVer : UDINT;
		fb : REFERENCE TO AsArLogGetInfo;
	END_STRUCT;
END_TYPE
```

### Library Logical/Libraries/wbrServices/wbrMemSvc (ANSIC)
Depends on: AsMem

#### wbrMemSvc.typ - Exported data types
```iecst
(*** /*****************************************************************
 * \copyright -- Piedmont Automation
 ********************************************************************
 * Program : wbrMemSvc
 * \file :   wbrMemSvc.typ
 * \author : Blanton Radford
 * \date Created: April 14, 2016
 ********************************************************************
 * Data types of library wbrMemSvc
 ****************************************************************/ ****)

TYPE
	wbrMemSvcStatus_typ : 	STRUCT
		memInitValid : BOOL;
		blockFree : UDINT; (*Size of the largest available heap memory bock*)
	END_STRUCT;
	wbrMemSvcStoredConfig_typ : 	STRUCT
		memRequestSize : UDINT; (*Size of the heap memory partition to be requested during initialization*)
	END_STRUCT;
	wbrMemService_typ : {REDUND_UNREPLICABLE} 	STRUCT
		status : {REDUND_UNREPLICABLE} wbrMemSvcStatus_typ;
		config : REFERENCE TO wbrMemSvcStoredConfig_typ;
	END_STRUCT;
END_TYPE
```

### Library Logical/Libraries/wbrServices/wbrPingSvc (ANSIC)
Depends on: AsICMP, wbrLogSvc, bglibasWBR, AsTime

### bglibasWBR_C.h
```c
/********************************************************************
 * \copyright -- Piedmont Automation
 ********************************************************************
 * Program : wbrServices_C_Includes
 * \file :   bglibasWBR_C.h
 * \author : Blanton Radford
 * \date Created: August 17, 2015
 *******************************************************************/

#include <stdarg.h>

#include <bur/plctypes.h>

UDINT  bgSSMPrintToTextLog(struct bgSSM_typ* p, const char* format, ...);
```

### Library Logical/Libraries/wbrServices/wbrsprintf (ANSIC) - Writes user-formatted output to a string

#### ofmt.c
```c
/*
 *  __ofmt - in-memory text conversion and formatting
 *
 *  __ofmt is used by printf(), fprintf() and sprintf() to format
 *  a string.
 *
 *  A format argument is a string to be output with optional embedded
 *  conversion specifications.  The conversion specifications start with
 *  a `%' and end with a conversion character
 */

#include <stdarg.h>
#include <stdio.h>
#include <limits.h>
#include <ctype.h>
#include <string.h>
/*#include <introl.h>*/
#define FLOATS  /*!!!*/
#define LONGS /*!!!*/

extern void __cvtflasc(double arg, int ndigits, int *decpt, int *sign, char eflag, int bufsize, char *buf);

/* to save space on smaller processors, we will undef
 * all ctype macros, this will cause their functions to be used.
 */
#if defined __CC01__ || defined __CC03__ || defined __CC11__ || defined __CC09__
#undef isalnum
#undef isalpha
#undef iscntrl
#undef isdigit
#undef isgraph
#undef islower
#undef isprint
#undef ispunct
#undef isspace
#undef isupper
#undef isxdigit
#undef __tolower
#undef __toupper
#endif /* use less memory */

/*  LONGINTS will be defined if longs and ints are the same size
 *  on the target.
 */

#if INT_MAX == LONG_MAX
#define LONGINTS 1
#undef LONGS
#else
#define LONGINTS 0
#endif

/*
 * a few typedefs and defines
 */
#ifdef UCHAR
#undef UCHAR
#endif
typedef unsigned char UCHAR;
#ifdef UINT
#undef UINT
#endif
typedef unsigned int UINT;
#ifdef ULONG
#undef ULONG
#endif
typedef unsigned long ULONG;
#ifdef ULLONG                                                                   //  WBR: added 2013-08-21  for future long long support
#undef ULLONG
#endif
typedef unsigned long long ULLONG;                                              //  WBR: added 2013-08-21  for future long long support

#define INITPREC  6 /* number + (opt sign) */
#define MAXLEN 21

static void putcurrent(FILE *stream, char **line, /*int buf_size,*/ int putvalue, int *numberput);

/*
 * definitions for __ofmt flags.
 */
#define INTPAD    0x01
#define LEFTJUST  0x02  /* left justify output */
#define ALTERNATE 0x04  /* use "#" alternate form */
#define LONGFLAG  0x08  /* is this a long argument */
#define SIGNFLAG  0x10  /* must we output a sign */
#define LEADINGZERO 0x20  /* output a leasing zero */
#define PRECISIONFLAG 0x40  /* user specified precision */

#define FLOATFLAG 0x01  /* are we in a float format */
#define DECIMALPOINT  0x02  /* should we output a decimalpoint */
#define EXPSIGN   0x04  /* sign of exponent 0:+, 1:- */
#define EXPONENT  0x08  /* exponent: yes or no */
#define ETYPE   0x10  /* "e" format conversion in __cvtflasc */

int bf_sz;

int __ofmt(FILE *stream, char *line, int buf_size, const char *format, va_list ap)      // WBR: added buf_size
  {
  UCHAR flags;    /* flag holder for output formatting */
  UCHAR fflags;   /* flags for float formatting */
  char  work[MAXLEN]; /* Maximum character length or any float, int, etc. */
  char  *workptr; /* temp pointer used to move through work[] */
  char  c;    /* current character in format string */
  char  base;   /* base for numerical conversions */
  char  sign;   /* (+,-, ,\0) used when SIGNFLAG is set */
  int width;    /* %3: format width: default 0 */
  int precision;  /* %.3: format precision: default -1 */
  int numberput = 0;  /* number of characters output */
  char  pad;    /* character to pad fields with */
  int totallength;  /* Number of spaces to pad determined in each case */
  int numchars; /* number of characters in 'number' */
#ifdef  LONGS
  long  ltemp;    /* long temporary */
  ULONG conv_val; /* variable used by 'convert:' which contains the number */
#else
  int ltemp;    /* int temporary */
  UINT  conv_val; /* variable used by 'convert:' which contains the number */
#endif
  long long lltemp;   // long long temporary                                    WBR: added 2013-08-21  for future long long support
  ULLONG    conv_llval;
  int decpt = 0;  /* double decimal point (needed anyway) */
#ifdef  FLOATS
  int exponent; /* represents the exponent value */
  double  ftemp;    /* double temporary */
  int exponent_begin; /* beginning index into "work[]" for the exponent */
#endif

bf_sz=  buf_size;     // WBR: set buffer size for wbrsnprintf

  while ((c = *format)) /* get a format character */
    {
    if (c != '%') /* if no conversion specifier ... */
      {
      /* just send character */
      putcurrent(stream, &line, c, &numberput);
      ++format;
      continue; /* and try again */
      }

    workptr = work;   /* set up work buffer ptr */
    fflags = flags = 0; /* initial all flag bits to 0 */
    precision = -1;
    width = 0;
    pad = ' ';    /* default padding character */

incloop:  ++format;
loop:   switch (c = *format)
      {
      case ' ':
        flags |= SIGNFLAG;
        sign = ' ';
        goto incloop;
      case '#':
        flags |= ALTERNATE;
        goto incloop;
      case '-':
        flags |= LEFTJUST;
        goto incloop;
      case '+':
        flags |= SIGNFLAG;
        sign = '+';
        goto incloop;
      case '%':
        putcurrent(stream, &line, '%', &numberput);
        ++format;
        break;
      case '0':
        /* set pad character to zero */
        pad = '0';
        goto incloop;
#if defined(LONGS) || defined(LONGINTS)
      case 'l':
        flags |= LONGFLAG;
        goto incloop;
#endif /* LONGFLAGS */
      case '*':
        /* get width */
        width = (va_arg(ap, int));
        if (*(++format) != '.')
          goto loop;
        ++format;
        if (isdigit(*format))
          goto numprecision;
        if (*format != '*')
          goto loop;
argprecision:
        flags |= PRECISIONFLAG;
        precision = va_arg(ap, int);
        goto incloop;
      case '1': case '2': case '3':
      case '4': case '5': case '6':
      case '7': case '8': case '9':
        while(isdigit(*format))
          width = 10 * width + (*(format)++ - '0');
        if (*format == '.')
          {
      case '.':
          /* get the maximum width allowed
           */
          flags |= PRECISIONFLAG;
          precision = 0;
          ++format; /* skip the '.' */

          if (*format == '*')
            goto argprecision;
          else
numprecision:
            while (isdigit(*format))
              precision = 10 * precision +
              (*(format)++ - '0');
          }
        goto loop;
#ifdef  FLOATS
      {
      int negative;

      case 'G':
      case 'g':
        ftemp = (va_arg(ap,double));
        __cvtflasc(ftemp, precision, &decpt, &negative,
          0, sizeof(work), workptr);
        if (decpt < -4 && decpt < precision)
          goto float_common;
        goto set_e_flags;
      case 'E':
      case 'e':
        /* set the E format flag and other float flags */
        ftemp = (va_arg(ap,double));
      set_e_flags:
        fflags |= EXPONENT | ETYPE;
        goto float_common;
      case 'F':
      case 'f':
        ftemp = (va_arg(ap,double));
      float_common:
        fflags |= FLOATFLAG;
        exponent = 0;
        workptr = work;

        if (precision == -1)
          precision = INITPREC;

        __cvtflasc(ftemp, precision, &decpt, &negative,
          fflags & ETYPE, sizeof(work), workptr);

        if (precision != 0)
          fflags |= DECIMALPOINT;

        if (negative)
          {
          flags |= SIGNFLAG;
          sign = '-';
          }

        if (decpt < 0)
          flags |= LEADINGZERO;
        else
          flags &= ~LEADINGZERO;

        if (fflags & EXPONENT)
          {
          if (decpt < 0)
            {
            fflags |= EXPSIGN;
            decpt = -decpt;
            exponent = decpt + 1;
            }
          else
            {
            exponent = decpt - 1;
            fflags &= ~EXPSIGN;
            }
          decpt = 1;
          workptr[MAXLEN-1] = '\0';
          if (exponent > -10 && exponent < 10)
            {
            workptr[MAXLEN-2] = exponent + '0';
            workptr[MAXLEN-3] = '0';
            exponent = 4;
            exponent_begin = MAXLEN - 3;
            }
          else if (exponent > -100 && exponent < 100)
            {
            workptr[MAXLEN-2] = exponent % 10 + '0';
            workptr[MAXLEN-3] = (exponent / 10) % 10 + '0';
            exponent = 4;
            exponent_begin = MAXLEN - 3;
            }
          else
            {
            char *s = workptr + MAXLEN - 1;
            int tmp;
            for (tmp = 0 ; tmp < 3 ; ++tmp)
              {
              *--s = exponent % 10 + '0';
              exponent /= 10;
              }
            exponent = 5;
            exponent_begin = MAXLEN - 4;
            }
          }

        if (decpt > 0)
          totallength = decpt;
        else
          totallength = 1;

        totallength += precision + totallength +
          ((fflags & DECIMALPOINT) != 0) + ((flags & SIGNFLAG) != 0);

        goto output;  /* output */
      }
#endif
      case 'N':
      case 'n':
        *(va_arg(ap, int *)) = numberput;
        continue;
      case 'I':
      case 'i':
      case 'D':
      case 'd':
        /* convert signed `int' or `long' to decimal
         */
#ifdef  LONGS
        if (flags & LONGFLAG)
          {
          ltemp = (va_arg(ap, long));
          if (ltemp < 0)
            {
            flags |= SIGNFLAG;
            ltemp = -ltemp;
            sign = '-';
            }
          }
        else
#endif
          {
          ltemp = (va_arg(ap, int));
          if (ltemp < 0)
            {
            flags |= SIGNFLAG;
            sign = '-';
            ltemp = -ltemp;
            }
          }

        conv_val = ltemp;
        base = 10;
        goto convert;

      case 'U':
      case 'u':
        /* convert unsigned instead of signed
         */
#ifdef  LONGS
        if (flags & LONGFLAG)
          conv_val = (va_arg(ap,unsigned long));
        else
#endif
          conv_val = (va_arg(ap,unsigned));

        /* clear signflag
         */
        flags &= ~SIGNFLAG;
        base = 10;
        goto convert;

      case 'P':
      case 'p':
      case 'X':
      case 'x':
        /* convert to hexadecimal instead of decimal
         */
#ifdef  LONGS
        if (flags & LONGFLAG)
          conv_val = (va_arg(ap,unsigned long));
        else
#endif
          conv_val = (va_arg(ap,unsigned));
        base = 16;
        flags &= ~SIGNFLAG;
        goto convert;

      case 'O':
      case 'o':
        /* convert to octal instead of decimal
         */
#ifdef  LONGS
        if (flags & LONGFLAG)
          conv_val = (va_arg(ap,unsigned long));
        else
#endif
          conv_val = (va_arg(ap,unsigned));

        base = 8;
        flags &= ~SIGNFLAG;
        goto convert;

        /* convert - convert the value to the given
         * base and advance all the pointers
         */
      convert:
        {
        int val;
        char *v, *x, y, letter;

        numchars = 1;
        letter = (c == 'X' ? 'A' : 'a');
        val = conv_val % base;
        *workptr++ = val < 10 ? val + '0' : val + letter - 10;

        /* convert the string backwards and then reverse it
         */
        while ( ( conv_val = (conv_val / base) ) )/* changed parentheses order - 20100517 DFB */
                            /* originally  'while ((conv_val = conv_val)  / (base))' */
          {
          val = conv_val % base;                 /* get lowest digit */
          *workptr++ = (val < 10 ? val + '0' : val + letter - 10);
          ++numchars;
          }

        /* if alternate is set, use 'c' to determine which prefix
         * to output
         */
        if (flags & ALTERNATE)
          switch (c)
            {
            case 'x':
              *workptr++ = 'x';
              ++numchars;
              goto addthe0;
            case 'X':
              *workptr++ = 'X';
              ++numchars;
              goto addthe0;
            case 'o':
            case 'O':
addthe0:
              *workptr++ = '0';
              ++numchars;
              break;
            }
        *workptr = '\0';  /* terminate work buffer */

        /* reverse the string
         */
        for (v = work ,  x = v + numchars ; v < x ; )
          {
          y = *v;
          *v++ = *--x;
          *x = y;
          }

        flags &= ~LEADINGZERO;
        fflags &= ~(DECIMALPOINT | EXPONENT);

        if (precision && !width)
          width = precision;
        if (!(flags & PRECISIONFLAG))
          precision = numchars;
        else if (numchars <= precision && width <= precision)
          pad = '0';
        totallength = numchars + ((flags & SIGNFLAG) != 0);
        }
        goto output;
      case 'C':
      case 'c':
        /* send a character
         */
        *workptr++ = (va_arg(ap, int));
        *workptr = '\0';  /* terminate work buffer */
        numchars = totallength = precision = 1;
        goto output;

      case 'S':
      case 's':
        /* send a string
         */
        workptr = (va_arg(ap, char *));

        numchars=totallength=strlen(workptr);

        if ((flags & PRECISIONFLAG) && precision < totallength)
          totallength = precision;
        else
          precision = totallength;

        if (totallength > width)
          {
          numchars = totallength;
          width =  totallength;
          }

        /* fall into output, but don't overwrite "workptr" */
        goto output1;
      output:
        workptr = work; /* point to work buffer */
      output1:

        if (!(flags & LEFTJUST))
          {
          int i;

          for (i = width - (totallength < precision ? precision : totallength) ; i > 0 ; --i)
            putcurrent(stream, &line, pad ,&numberput);
          for (i = precision - totallength; i > 0 ; i--)
            putcurrent(stream, &line, '0' ,&numberput);
          }

        /* send out leading padding character
         */
        if (flags & SIGNFLAG)
          putcurrent(stream, &line, sign, &numberput);

        /* transfer the work buffer to the line
         */
#ifdef FLOATS
        if (fflags & FLOATFLAG)
          {
          if (decpt > 0)
            do
              {
              putcurrent(stream, &line,*workptr++,&numberput);
              }
            while (--decpt > 0);
          else
            putcurrent(stream, &line,'0',&numberput);

          if (fflags & DECIMALPOINT)
            putcurrent(stream, &line,'.',&numberput);
          while(decpt < 0 && precision > 0)
            {
            putcurrent(stream, &line,'0',&numberput);
            ++decpt;
            --precision;
            }

          while (precision > 0)
            {
            putcurrent(stream, &line,*workptr++,&numberput);
            --precision;
            }

          if (fflags & EXPONENT)
            {
            char *s;
            int i;

            putcurrent(stream, &line,'e',&numberput);
            if (fflags & EXPSIGN)
              putcurrent(stream, &line, '-', &numberput);
            else
              putcurrent(stream, &line, '+', &numberput);
            for ((s = &work[exponent_begin]); (i = *s) ; ++s)
               putcurrent(stream, &line, i, &numberput);
            }
          }
        else
#endif
          {
          int i;
          if (!precision || numchars < precision)
            i = numchars;
          else
            i = precision;
          for ( ; i ; --i)
            putcurrent(stream, &line,*workptr++,&numberput);
          }
        /* if left justified, pad on the right
         */
        if (flags & LEFTJUST)
          {
          int i;

          for (i = width - totallength; i > 0 ; i--)
            /* here always pad with spaces */
            putcurrent(stream, &line, ' ', &numberput);
          }
        ++format;
        break;

      default:
        /* if the character after the `%' wasn't a
         * null then add it to the print buffer and
         * increment `format'
         */
        if (*format)
          putcurrent(stream, &line, *format++, &numberput);
      }
    }
  /* terminate line */
  putcurrent(stream, &line, '\0', &numberput);
  return numberput - 1;
  }

static void putcurrent(FILE *stream, char **line, int putvalue, int *numberput)
  {
  (*numberput)++;
  if((stream == NULL) && ((*numberput < bf_sz) || (putvalue == '\0')))         // WBR: added size check for snprintf function
    *(*line)++ = putvalue;
  else
    /*putc(putvalue,stream)*/;
  }
```

#### wbrsprintf.c
```c
/*
 *      sprintf - write a printf-formatted string to memory at "line"
 */

#include <stdarg.h>
#include <stdio.h>
#include <limits.h>

#include "wbrsprintf.h"
// #include "sprintf_s.h"

int __ofmt(FILE *stream, char *line, int buf_size,
                                     const char *format, va_list ap);

int wbrvsprintf(char *s, const char *fmt, va_list ap)
{
 int num;

  return num = __ofmt(0, s, INT_MAX, fmt, ap);
}

int wbrvsnprintf(char *s, int buf_size, const char *fmt, va_list ap)
{
 // int num;

  // return num = __ofmt(0, s, buf_size, fmt, ap);
  return __ofmt(0, s, buf_size, fmt, ap);
}

int wbrsprintf(char *s, const char *fmt, ...)
{
 int num;
 va_list ap;

  va_start(ap, fmt);
  num = wbrvsprintf(s, fmt, ap);
  va_end(ap);
  return num;
}

int wbrsnprintf(char *s, int buf_size, const char *fmt, ...)
{
 int num;
 va_list ap;

  va_start(ap, fmt);
  num = wbrvsnprintf(s, buf_size, fmt, ap);
  va_end(ap);
  return num;
}
```

- Library Logical/Libraries/wbrServices/wbrSvcUtilities/wbrFltUtil (ANSIC) - Utilities for floating-point numbers.  Most return or act on double types, some on float types. (no source held here)

### Library Logical/Application/Creaser

#### LocalFunctions.fun
```iecst
FUNCTION_BLOCK PulseTrain (*TODO: Add your comment here*) (*$GROUP=User,$CAT=User,$GROUPICON=User.png,$CATICON=User.png*)
	VAR_INPUT
		TimeOn : TIME;
		TimeOff : TIME;
	END_VAR
	VAR_OUTPUT
		bFlashOut : BOOL;
	END_VAR
	VAR
		bFlashTrig : BOOL;
		TP_FLASH : TP;
		MaxTime : TIME;
	END_VAR
END_FUNCTION_BLOCK
```

#### Action_Manage_Update_Total_Runtime.st
```iecst
ACTION Action_Manage_Update_Total_Runtime:

	IF bgTimerIsTimeOut(Timer_Total_Runtime) THEN
		gStatistics.total_runtime := gStatistics.total_runtime + 1;
		bgTimerStart(Timer_Total_Runtime, 1000);

		gStatistics.runtime_h := gStatistics.total_runtime / 3600;
		gStatistics.runtime_m := (gStatistics.total_runtime 	/ 60) MOD 60;
		gStatistics.runtime_s := gStatistics.total_runtime MOD 60;
	END_IF;

	bgTimerCyclic(Timer_Total_Runtime);

END_ACTION
```

#### Action_Stop_Feeder.st
```iecst
ACTION Action_Stop_Feeder:
	AxisControl.MoveVelocity := FALSE;
	AxisControl.MoveAbsolute := FALSE;
	AxisControl.MoveAdditive := FALSE;
	AxisControl.Stop := FALSE;
	AxisControl();

	AxisPar.Velocity := gRecCfg.active.Cfg.Creaser.PreInsertSpeed;
	AxisPar.Acceleration := gRecCfg.active.Cfg.Creaser.FeedAxisAccel;
	AxisPar.Deceleration := gRecCfg.active.Cfg.Creaser.FeedAxisDecel;

	AxisControl.Stop := TRUE;
	AxisControl();
END_ACTION
```

#### Action_Validate_Board_Length.st
```iecst
ACTION Action_Validate_Board_Length:

	length_calculated_total := 0;
	flagBoardLengthCfgErr := FALSE;

	FOR ii_crease_count := 0 TO gRecCfg.active.Rec.Crease.CreaseCount - 1 BY 1 DO

		length_calculated_total := length_calculated_total + gRecCfg.active.Rec.Crease.CreaseDistance_mm[ii_crease_count] + gRecCfg.active.Rec.Crease.CreaseWidth_mm;

	END_FOR;

	IF length_calculated_total > (gRecCfg.active.Rec.Crease.TotalBoardLength + gRecCfg.active.Cfg.Creaser.BoardLengthTolerance) THEN
		gAlarms.Board_Length_GT_Confgd_Amount := TRUE;
		flagBoardLengthCfgErr := TRUE;
//	ELSIF length_calculated_total < (gRecCfg.active.Rec.Crease.TotalBoardLength - gRecCfg.active.Cfg.Creaser.BoardLengthTolerance) THEN
//		gAlarms.Board_Length_LT_Confgd_Amount := TRUE;
//		flagBoardLengthCfgErr := TRUE;
	END_IF;

END_ACTION
```

#### Main.st
```iecst
PROGRAM _INIT

	Action_Init_Infeed_Axis; //Set pointer values/initialize servo drive FBK MpAxisBasic instance

	MachineState := MACHINE_STATE_INIT;

	Pulse_Slow.TimeOn := DEFINE_SLOW_PULSE_PERIOD;
	Pulse_Slow.TimeOff := DEFINE_SLOW_PULSE_PERIOD;

	Pulse_Fast.TimeOn := DEFINE_FAST_PULSE_PERIOD;
	Pulse_Fast.TimeOff := DEFINE_FAST_PULSE_PERIOD;

END_PROGRAM

PROGRAM _CYCLIC

	IF gStatistics.Reset THEN //Reset all statistics
		brsmemset(ADR(gStatistics), 0, SIZEOF(Global_Statistics_typ)); //Kind of a weird way to do this- essentially just writes 0's to the entirety of the memory the structure occupies (thus "zeroing-out" the counters)
	END_IF;

	Action_Eval_ErrorState_Statuses; //Evaluate the conditions that put machine into ERR state

	//Eval conditions that would send the machine into ERR state if the machine isn't already in ERR or INIT state->

	IF EDGEPOS(IO.iSafeMachineState) OR iMachineErrorReset THEN
		ProcessState := PRCS_STATE_INIT;
		gAlarmResetRequested := TRUE;
		//		gStatistics.Reset := TRUE;
		MachineState := MACHINE_STATE_INIT;
	END_IF;

	IF EDGEPOS(MachineState = MACHINE_STATE_ERROR) THEN
		AxisControl.MoveVelocity := FALSE;
		AxisControl.MoveAbsolute := FALSE;
		AxisControl.MoveAdditive := FALSE;
		AxisControl.Stop := TRUE;
		AxisControl();
	END_IF;

	BoardEjectUIButton_Hide := BOOL_TO_USINT(NOT ((MachineState = MACHINE_STATE_IDLE OR MachineState = MACHINE_STATE_MANUAL_EJECT) AND IO.iFiberOpticSensor));

	StartUIButton_Hide := NOT (MachineState = MACHINE_STATE_IDLE);
	StopUIButton_Hide := NOT (MachineState = MACHINE_STATE_RUNNING);

	CASE MachineState OF
		MACHINE_STATE_INIT:
			IO.oBoardFeedingLight := FALSE;
			IO.oUIIndicatorLight := FALSE;
			AxisControl.Power := FALSE;

			MachineState := MACHINE_STATE_HARDWARE_INIT;

		MACHINE_STATE_HARDWARE_INIT:
			IO.oBoardFeedingLight := FALSE;
			IO.oUIIndicatorLight := FALSE;

			IF AxisControl.Info.ReadyToPowerOn THEN
				AxisControl.Power := TRUE;
				MachineState := MACHINE_STATE_AXIS_POWER;
			END_IF;

		MACHINE_STATE_AXIS_POWER:
			IO.oBoardFeedingLight := FALSE;
			IO.oUIIndicatorLight := FALSE;

			IF AxisControl.PowerOn THEN
				Action_Stop_Feeder;
				MachineState := MACHINE_STATE_IDLE;
			END_IF;

		MACHINE_STATE_IDLE:
			IO.oBoardFeedingLight := FALSE;
			IO.oUIIndicatorLight := Pulse_Slow.bFlashOut;

			IF EDGEPOS(iManualBoardEject) THEN

				AxisControl.MoveVelocity := FALSE;
				AxisControl.MoveAbsolute := FALSE;
				AxisControl.MoveAdditive := FALSE;
				AxisControl.Stop := FALSE;
				AxisControl();

				AxisPar.Velocity := gRecCfg.active.Rec.FeedVelocity;
				AxisPar.Acceleration := gRecCfg.active.Cfg.Creaser.FeedAxisAccel;
				AxisPar.Deceleration := gRecCfg.active.Cfg.Creaser.FeedAxisDecel;

				AxisControl.MoveVelocity := TRUE;
				AxisControl();

				MachineState := MACHINE_STATE_MANUAL_EJECT;
			END_IF;

			IF EDGEPOS(iStartCommand) THEN
				IF IO.iFiberOpticSensor THEN
					gAlarms.Fiber_Optic_Blocked_RunCmd := TRUE;
					MachineState := MACHINE_STATE_ERROR;
				ELSIF NOT IO.iCreaserShaftSensor THEN
					gAlarms.Manual_Home_Creaser_Blade := TRUE;
					MachineState := MACHINE_STATE_ERROR;
				ELSE
					//					setflagCreaserIndexCommand := TRUE;

					Action_Start_Feeder;
					ProcessState := PRCS_STATE_INIT;
					MachineState := MACHINE_STATE_RUNNING;
				END_IF;
			END_IF;

		MACHINE_STATE_MANUAL_EJECT:
			IO.oBoardFeedingLight := TRUE;
			IO.oUIIndicatorLight := Pulse_Slow.bFlashOut;

			IF (NOT IO.iFiberOpticSensor AND IO_LastCycle.iFiberOpticSensor) OR NOT iManualBoardEject THEN
				Action_Stop_Feeder;
				MachineState := MACHINE_STATE_IDLE;
			END_IF;

		MACHINE_STATE_RUNNING:
			IO.oUIIndicatorLight := TRUE;

			Action_Manage_Update_Total_Runtime;

			Action_Tally_Board_L;

			IF iSoftStopCommand THEN

				IF NOT (ProcessState = PRCS_STATE_SOFT_STOP) THEN
					Action_Stop_Feeder;
				END_IF;

				ProcessState := PRCS_STATE_SOFT_STOP;
			END_IF;

			Action_CreaserProcess_SM; //Crease motor <-> movement cycle <-> FiOS state machine

		MACHINE_STATE_ERROR: //ERROR state.  Note that this state is exited via the logic ABOVE the state machine.
			IO.oBoardFeedingLight := FALSE;
			IO.oUIIndicatorLight := Pulse_Fast.bFlashOut AND Pulse_Slow.bFlashOut;

			Current_Crease_Section_Length := 0;

			ProcessState := PRCS_STATE_INIT;

	END_CASE;

	Pulse_Slow;
	Pulse_Fast;

	Action_Creaser_Idx; //Reads/sets flag variables indicating current state of the creasing motor
	Action_AxisControl_Mgmt; //Calls Infeed Axis Control FBK, sets/resets drive errors

	IO_LastCycle := IO; //Latch previous cycle IO values (since EDGEPOS() has some weird caveats)
END_PROGRAM

PROGRAM _EXIT
	(* Insert code here *)

END_PROGRAM
```

#### PulseTrain.st
```iecst
(* TODO: Add your comment here *)
FUNCTION_BLOCK PulseTrain

	MaxTime := TimeOn + TimeOff ;
	TP_FLASH(IN:=bFlashTrig, PT:= (MaxTime + T#100ms));
	IF NOT bFlashTrig THEN
		bFlashTrig := TRUE;
	END_IF;

	IF (TP_FLASH.ET < TimeOn) THEN
		bFlashOut := TRUE;
	ELSIF (TP_FLASH.ET >= TimeOn) AND (TP_FLASH.ET <= MaxTime) THEN
		bFlashOut := FALSE;

	ELSE
		bFlashTrig := FALSE;
	END_IF;

END_FUNCTION_BLOCK
```

### Program Logical/Auxiliary_Services_Control/File_Handling

#### Cyclic.st
```iecst
PROGRAM _CYCLIC
	File_Manager_Control;
	File_Manager_UIConnect;

	Alarm_File;
	Alarm_File_UI();

END_PROGRAM
```

#### Init.st
```iecst
PROGRAM _INIT
	File_Manager_Control.MpLink := ADR(File_Manager_MpLink);
	File_Manager_Control.Enable := TRUE;
	File_Manager_Control.UIConnect := ADR(File_Manager_UIConnect);

	File_Manager_UIConnect.DeviceList.DeviceNames[0] := 'ROOT';
	File_Manager_UIConnect.DeviceList.DeviceNames[1] := 'Config';
	File_Manager_UIConnect.DeviceList.DeviceNames[2] := 'Recipe';
	File_Manager_UIConnect.DeviceList.DeviceNames[3] := 'Process';
	File_Manager_UIConnect.DeviceList.DeviceNames[4] := 'USB1';
	File_Manager_UIConnect.DeviceList.DeviceNames[5] := 'USB2';

	File_Manager_Control.UISetup.FileListSize := 8;
	File_Manager_Control.UISetup.FileListScrollWindow := 5;

	File_Manager_Control;

	Alarm_File_UI.MpLink := ADR(File_Manager_MpLink);
	Alarm_File_UI.Enable := TRUE;
	Alarm_File_UI.Mode := mpALARM_BASIC_UI_MODE_ALL;

	Alarm_File_UI.UISetup.ImageSize := 20;
	Alarm_File_UI.UISetup.AlarmImage := ADR(Alarm_File.AlarmImage[0]);
	Alarm_File_UI.UISetup.AcknowledgeImage := ADR(Alarm_File.AcknowledgeImage[0]);
	Alarm_File_UI.UISetup.AddInfoStringSize := 100;
	Alarm_File_UI.UISetup.AddInfo := ADR(Alarm_File.AddInfo[0]);

	Alarm_File;
	Alarm_File_UI();

END_PROGRAM
```

### bgdebug.h
```c
#ifndef _BG_DEBUG_H
#define _BG_DEBUG_H

#ifdef WIN32
#define DBG printf
#define DBGMSG printf

#define DBGCRT printf
#define DBGERR printf
#define DBGWAR printf
#define DBGINF printf
#define DBGDBG printf

#else

#include <bur/plc.h>
#include "bgsprintf.h"
#include "bgringbuffer.h"

#define BG_DEBUG_LEVEL_CRITICAL		0
#define BG_DEBUG_LEVEL_ERROR		1
#define BG_DEBUG_LEVEL_WARNING		2
#define BG_DEBUG_LEVEL_INFO			3
#define BG_DEBUG_LEVEL_DEBUG		4

#define BG_DEBUG_UNUSED	0x0

/*
- To completly remove debug msgs from the source code use:
#define BG_DEBUG_ENABLE 0
*/
#define BG_DEBUG_ENABLE 1

/*ptr to global ring buffer for debug messages*/
_GLOBAL bgRingBuffer_typ gRingBuffer;

#if BG_DEBUG_ENABLE == 1
/*BG_DEBUG_ENABLE == 1 => debug messages present in the source code*/
#define DBG(format, args...)	bgRingBuffPutDbgInfo(&gRingBuffer, __FILE__, __FUNCTION__, BG_DEBUG_LEVEL_CRITICAL, BG_DEBUG_UNUSED, format, ## args);
#define DBGMSG(format, args...)	bgRingBuffPrintf(&gRingBuffer, format, ## args);

#define DBGCRT(format, args...)	bgRingBuffPutDbgInfo(&gRingBuffer, __FILE__, __FUNCTION__, BG_DEBUG_LEVEL_CRITICAL, BG_DEBUG_UNUSED, format, ## args);
#define DBGERR(format, args...)	bgRingBuffPutDbgInfo(&gRingBuffer, __FILE__, __FUNCTION__, BG_DEBUG_LEVEL_ERROR, BG_DEBUG_UNUSED, format, ## args);
#define DBGWAR(format, args...)	bgRingBuffPutDbgInfo(&gRingBuffer, __FILE__, __FUNCTION__, BG_DEBUG_LEVEL_WARNING, BG_DEBUG_UNUSED, format, ## args);
#define DBGINF(format, args...)	bgRingBuffPutDbgInfo(&gRingBuffer, __FILE__, __FUNCTION__, BG_DEBUG_LEVEL_INFO, BG_DEBUG_UNUSED, format, ## args);
#define DBGDBG(format, args...)	bgRingBuffPutDbgInfo(&gRingBuffer, __FILE__, __FUNCTION__, BG_DEBUG_LEVEL_DEBUG, BG_DEBUG_UNUSED, format, ## args);

#else
/*BG_DEBUG_ENABLE == 0 => all debug messages removed from the source code*/
#define DBG(format, args...)  ;
#define DBGMSG(format, args...)  ;

#define DBGCRT(format, args...)	;
#define DBGERR(format, args...)	;
#define DBGWAR(format, args...)	;
#define DBGINF(format, args...)	;
#define DBGDBG(format, args...)	;

#endif /*#if BG_DEBUG_ENABLE*/

#endif /*#ifdef WIN32*/

#endif /*#ifndef _BG_DEBUG_H*/
```

### bgfsig.h
```c
#ifndef _BG_FSIG_C
#define _BG_FSIG_C

int bgFileSignatureVerify(char *inFileBuffer, char *resultStringMinLen64);

#endif
```

### bgftpclient.h
```c
/*
File:
bgFtpClient.h

About:
------
- FTP (File Transfer Protocol) Client implementation for B&R PCC
*/
#ifndef _BG_FTPCLIENT_H
#define _BG_FTPCLIENT_H

#include <bur/plctypes.h>
#include <AsARCfg.h>
#include <ethsock.h>
#include <astcp.h>
#include "bgstatemachine.h"
#include "bgstring.h"

/*
Public data types:
-----------------
*/

/*User Private Library Error Numbers (value assigned as suggested in the B&R help file)*/
#define USER_ERROR_MIN  0xC350
#define USER_ERROR_MAX  0xEA5F
#define USER_ERROR_FTP  USER_ERROR_MIN + 10

#define CMD_DONE	0
#define CMD_BUSY	1
#define CMD_ERROR	2

typedef struct ftpClientUser_typ{
   	DINT cmd;
   	int dataType; /*asciiOrBinary*/
	char fileName[128];
	char *dataBuffer;
	int dataBufferLength;
    int disconnectRequest;
    int connectRequest;
}ftpClientUser_typ;

#define FTPCLIENT_RESPONSECODE_LEN 16

#define FTPCLIENT_CMDBUFSIZE	256

typedef struct bgFtpClient_typ{
	bgStateMachine_typ smFtp;
	bgStateMachine_typ smFtpCmd;
	bgStateMachine_typ smFtpMultiCmd;
	bgStateMachine_typ smCmdSocket;
	bgStateMachine_typ smDataSocket;

	unsigned int userState; 	/*state of the user command execution*/

	int	cmdError;
	int	cmdErrorCode;

	char isConnected;
	char isLoggedIn;
	char isDataPortReady;
	char isDoneMultiCmd;
	char isErrorMultiCmd;

	char sockData_Timer;
	int sockData_TimerTime;
	int sockData_TimerCounter;

	char serverResponseCode;

	DINT sock;			/*command socket*/
	DINT sockData;		/*data socket - listen*/
	DINT sockData01;	/*data socket - send/recv*/

	ETH_sockaddr_typ ftpServerAdrCmd;
	ETH_sockaddr_typ ftpServerAdrData;
	ETH_sockaddr_typ ftpClientAdrData;

	/*non-blocking I/O control*/
	ETH_fd_set_typ fdR;
	ETH_fd_set_typ fdW;
	ETH_timeval_typ timeOut;

	char cmdSendBuf[FTPCLIENT_CMDBUFSIZE];
	char cmdRecvBuf[FTPCLIENT_CMDBUFSIZE];
#if 0
	char dataSendBuf[1024];
	char dataRecvBuf[1024];
#endif
	char cmdExpectedServerResponse[FTPCLIENT_RESPONSECODE_LEN];
	char cmdExpectedServerResponseCodeOrString; /*0-code,1-string*/

	DINT sendLen;
	DINT recvLen;
	DINT sendLenData;
	DINT recvLenData;

	TcpOpen_typ TCPopen_1;
	TcpServer_typ TCPserv_1;
	TcpSend_typ TCPsend_1;
	TcpRecv_typ TCPrecv_1;
	TcpClose_typ TCPclose_1;
	CfgGetIPAddr_typ CfgIPAddr_1;
	char CfgIPAddrString[20];
	unsigned int ipAddr[4];	/*client's own ip address; i.e. 192.168.1.6 -> ipAddr[0]=192, ipAddr[1]=168, etc*/

	int counter;
	int dataPort;
	bgStringList_typ responseList;
	int test;
	ftpClientUser_typ user;
	char 	*rxDataBuff;
}bgFtpClient_typ;

/*
Public functions:
-----------------
*/
void bgFtpClientCyclic(bgFtpClient_typ *p, int msgId);

void bgFtpClientDisconnect(bgFtpClient_typ *p);

void bgFtpClientConnectAndLogin(bgFtpClient_typ *p, char *ethernetInterface, char *serverIp);
int bgFtpClientIsLoggedIn(bgFtpClient_typ *p);
int bgFtpClientIsConnected(bgFtpClient_typ *p);
int bgFtpClientIsError(bgFtpClient_typ *p);

void bgFtpClientCmdCwdInit(bgFtpClient_typ *p, char *fileName, char *buffer, int bufferLength);
int bgFtpClientCmdCwdOnDone(bgFtpClient_typ *p);
int bgFtpClientCmdCwdOnError(bgFtpClient_typ *p);

void bgFtpClientCmdGetFileInit(bgFtpClient_typ *p, char *fileName, char* buffer, int bufferLength);
int bgFtpClientCmdGetFileOnDone(bgFtpClient_typ *p);
int bgFtpClientCmdGetFileOnError(bgFtpClient_typ *p);

void bgFtpClientCmdListInit(bgFtpClient_typ *p, char *buffer, int bufferLength);
int bgFtpClientCmdListOnDone(bgFtpClient_typ *p);
int bgFtpClientCmdListOnError(bgFtpClient_typ *p);

void bgFtpClientCmdPwdInit(bgFtpClient_typ *p, char *buffer, int bufferLength);
int bgFtpClientCmdPwdOnDone(bgFtpClient_typ *p);
int bgFtpClientCmdPwdOnError(bgFtpClient_typ *p);

#endif
```

### bgHttpAppXmlRpc.h
```c
#ifndef _bgHttpAppXmlRpc_h_
#define _bgHttpAppXmlRpc_h_

#include "bgTcpSocketClientServer.h"
#include "bgXmlRpcParser.h"

typedef struct httpAppXmlRpc_typ{
/*Note: following object(s) require(s) external ("allocated") memory!*/

bgXmlRpcParser_typ xmlRpcData;

}httpAppXmlRpc_typ;

void bgXmlRpcServerApplication(bgTcpSocketSession_typ* pSession);
int bgXmlRpcServerAppCommon(bgTcpSocketSession_typ* pSession);
int bgXmlRpcServerSendFaultResponse(bgTcpSocketSession_typ* pSession, int faultCode, char* faultString);
int bgXmlRpcServerSendResponse(bgTcpSocketSession_typ* pSession, char* pContent, int contentSize);

void bgXmlRpcClientSetConnection(bgTcpSocketClient_typ* pClient, char* serverIpAddr, int serverPortNumber);
void bgXmlRpcClientSendRequest(bgTcpSocketClient_typ* pClient, char* pContent , int contentSize);
void bgXmlRpcClientApplication(bgTcpSocketSession_typ* pSession);

#endif
```

### bgHttpProtocol.h
```c
#ifndef _bgHttpProtocol_h_
#define _bgHttpProtocol_h_

#include "bgTcpSocketClientServer.h"

#define APNDCL(line)	bgHttpSendBufApndContentLine(pSession, line)

void bgHttpServerSessionHandler(bgTcpSocketSession_typ* pSession);
void bgHttpClientSessionHandler(bgTcpSocketSession_typ* pSession);

void bgHttpSendErrorResponse(bgTcpSocketSession_typ* p, int responseCode);
void bgHttpServerSendResponse(bgTcpSocketSession_typ* pSession, int responseCode, char* pContent , int contentSize, char* contentType);
void bgHttpServerSendResponseBeg(bgTcpSocketSession_typ* pSession, int responseCode, char* contentType);
void bgHttpServerSendResponseEnd(bgTcpSocketSession_typ* pSession);

void bgHttpSendData(bgTcpSocketSession_typ* pSession);

char* bgHttpGetContentStartAddr(bgTcpSocketSession_typ* p);
int bgHttpGetContentLength(bgTcpSocketSession_typ* p);

void bgHttpClientSetConnection(bgTcpSocketClient_typ* pClient, char* serverIpAddr, int serverPortNumber);
void bgHttpClientSendRequest(bgTcpSocketClient_typ* pClient, char* pCmd, char* pContent , int contentSize, char* contentType);
void bgHttpClientSendRequestSetHeader(bgTcpSocketSession_typ* p, char* pCmd, int contentSize, char* contentType);

#endif
```

### bgBufMemAlloc.c
```c
#ifndef _BG_BUFMEMALLOC_C
#define _BG_BUFMEMALLOC_C

#include "bgBufMemAlloc.h"
//#include "string.h"

/*
##################################################################################
Buffer memory allocation
##################################################################################
*/
void bgBufMemAllocInit(bgBufMemAlloc_typ* p, char* pBufMem, int lengthBufMemBytes)
{
int i;

	p->pBufMem = pBufMem;
	p->lengthBufMemBytes = lengthBufMemBytes;
	p->lengthUsedMemBytes = 0;
	p->countUsedBlocks = 0;
	p->countMaxBlocks = BGBUFMEMALLOC_MAX_BLOCKS;
	for(i=0; i < p->countMaxBlocks; i++){
		p->memBlock[i].used = 0;
		p->memBlock[i].pMemBlock = 0;
		p->memBlock[i].lengthMemBlockBytes = 0;
	}
}

int bgBufMemAllocCreateBlock(bgBufMemAlloc_typ* p, int blockSize, char** pMemBlock, int* sizeMemBlock)
{
int i;
int availableBufMem = p->lengthBufMemBytes - p->lengthUsedMemBytes;

	if(blockSize >= availableBufMem)
		goto errorExit;

	if(p->countUsedBlocks >= p->countMaxBlocks)
		goto errorExit;

	for(i=0; i < p->countMaxBlocks; i++){
		if(!p->memBlock[i].used){
			p->memBlock[i].used = 1;
			p->memBlock[i].pMemBlock = (p->pBufMem + p->lengthUsedMemBytes);
			/*0 block size - use all available memory*/
			if(!blockSize)
				blockSize = availableBufMem;
			p->memBlock[i].lengthMemBlockBytes = blockSize;
			p->lengthUsedMemBytes += blockSize;
			p->countUsedBlocks++;
			if(pMemBlock)
				*pMemBlock = p->memBlock[i].pMemBlock;
			if(sizeMemBlock)
				*sizeMemBlock = p->memBlock[i].lengthMemBlockBytes;
			return 0;
		}
	}

errorExit:
	if(pMemBlock)
		*pMemBlock = 0;
	if(sizeMemBlock)
		*sizeMemBlock = 0;
	return 1;
}

char* bgBufMemAllocGetBlockPtr(bgBufMemAlloc_typ* p, int blockId, int* blockSize)
{
	if(blockSize)
		*blockSize = 0;

	if((blockId < p->countMaxBlocks) && (!p->memBlock[blockId].used)){
		if(blockSize)
			*blockSize = p->memBlock[blockId].lengthMemBlockBytes;
		return	p->memBlock[blockId].pMemBlock;
	}

	return 0;
}

/*
##################################################################################
String heap
##################################################################################
*/
char* bgStringHeapInit(bgStringHeap_typ* pHeap, char* pHeapMem, int memSize)
{
	pHeap->pMemStart = pHeapMem;
	pHeap->pMemCurrent = pHeap->pMemStart;
	*pHeap->pMemCurrent = 0;
	pHeap->memSize = memSize;
	pHeap->memFree = pHeap->memSize;
	return pHeap->pMemStart;
}

char* bgStringHeapAddString(bgStringHeap_typ* pHeap, char* pStr)
{
int len = strlen(pStr);
char* pCurString = pHeap->pMemCurrent;;

	/*adjust lentgh for 0 termination*/
	len += 1;

	if( len >= pHeap->memFree )
		return 0;

	strcpy(pCurString, pStr);

	/*move current ptr*/
	pHeap->pMemCurrent += len;

	/*reduce free mem*/
	pHeap->memFree -= len;

	return pCurString;
}
#endif
```

### bgDataStructures.c
```c
#ifndef _BG_DATASTRUCTURES_C
#define _BG_DATASTRUCTURES_C

#include "bgDataStructures.h"

#ifdef WIN32
#include <stdio.h>
#define DBGMSG printf
#else
#include "bgdebug.h"
#endif

#ifdef WIN32
static char* pTabs[30]={
"",
"    ",
"        ",
"            ",
"                ",
"                    ",
"                        ",
"                            ",
"                                ",
"                                    ",
"                                        ",
"                                            ",
"                                                ",
"                                                    ",
"                                                        ",
"                                                            ",
"                                                                ",
"                                                                    ",
};

static char* pStackDepth[30]={
" ",
"=",
"==",
"===",
"====",
"=====",
"======",
"=======",
"========",
"=========",
"==========",
"===========",
"============",
"=============",
"==============",
"===============",
"================",
"=================",
"==================",
};
#endif

/*
##################################################################################
Stack
##################################################################################
*/
void bgStackInit(bgStack_typ* stack)
{
    stack->index = 0;
}

char* bgStackPush(bgStack_typ* stack, char* data)
{
    if(stack->index >= BGSTACK_DEPTH_MAX)
		return 0;
/*
    printf("[%2d]push:%s\n", (int)data, pStackDepth[stack->index]);
*/
    stack->data[stack->index] = data;
    stack->index++;

	return data;
}

char* bgStackPop(bgStack_typ* stack)
{
    if(!stack->index)
        return 0;

    stack->index--;
/*
    printf("[%2d]pop :%s\n", (int)(stack->data[stack->index]), pStackDepth[stack->index]);
*/
    return stack->data[stack->index];
}

char* bgStackPeek(bgStack_typ* stack)
{
    if(!stack->index)
        return 0;

    return stack->data[stack->index - 1];
}

int bgStackGetItemCount(bgStack_typ* stack)
{
    return stack->index;
}

/*
##################################################################################
Tree  of Nodes (Each nodes has lf,rt,up,dw connections - 4C(onnections) nodes)
##################################################################################
*/
void bgTree4CInit(bgTree4C_typ* tree, char* pTreeMem, int treeMemSize)
{
int i;
bgTree4CNode_typ* node;

	if(!pTreeMem || (treeMemSize < 256) ){
		DBGMSG("bgTree4CInit: not enough memory!\n");
		tree->nodeCountMax = 0;
		return;
	}

	tree->nodeCountMax = treeMemSize / sizeof(bgTree4CNode_typ);
#ifdef WIN32
	DBGMSG("bgTree4CInit: max. number of nodes=%d\n", tree->nodeCountMax);
#endif
	tree->nodeCountUsed = 0;
	tree->nodes = (bgTree4CNode_typ*)pTreeMem;
	for(i=0; i<tree->nodeCountMax;i++){
        node = &tree->nodes[i];
        node->id = i;
		node->nodeCountMax = tree->nodeCountMax;
        bgTree4CNodeClr(node);
	}
}

void bgTree4CNodeClr(bgTree4CNode_typ* node)
{
	node->used = 0;
	node->up = 0;
	node->dw = 0;
	node->rt = 0;
	node->lf = 0;
	node->data = 0;
	node->dataType = 0;
}

bgTree4CNode_typ* bgTree4CNodeCreate(bgTree4C_typ* tree)
{
int i;
	if(!tree->nodeCountMax)
		return NULL;

	if( tree->nodeCountUsed >= tree->nodeCountMax){
		return NULL;
	}

	for(i=0; i<tree->nodeCountMax;i++){
		if(tree->nodes[i].used == 0){
			tree->nodes[i].used = 1;
			tree->nodeCountUsed++;
			return &tree->nodes[i];
		}
	}
	return NULL;
}

int bgTree4CGetCountFreeNodes(bgTree4C_typ* tree)
{
	return (tree->nodeCountMax -  tree->nodeCountUsed);
}

bgTree4CNode_typ*  bgTree4CGetRootNode(bgTree4C_typ* tree)
{
    return &tree->nodes[0];
}

void bgTree4CNodeDelete(bgTree4C_typ* tree, bgTree4CNode_typ* node)
{
	if(!tree->nodeCountMax)
		return;

	if(node->used){
#ifdef WIN32
        DBGMSG("bgTree4CNodeDelete(): node deleted, id=%d\n", node->id);
#endif
        bgTree4CNodeClr(node);
		if( tree->nodeCountUsed )
			tree->nodeCountUsed--;
	}
}

bgTree4CNode_typ*  bgTree4CNodePreviousLevel(bgTree4CNode_typ* node1)
{
bgTree4CNode_typ* n1 = node1;
bgTree4CNode_typ* n2;
int i;

	if( !n1 )
		return 0;

	if( n1->lf)
		return n1->lf;

	if( !n1->up )
		return 0;

    for(i=0;i<node1->nodeCountMax;i++){
        n2 = n1->up;

        if( !n2 )
			return n1->lf;

		n1 = n2;
    }

	return 0;
}

void bgTree4CNodeAddDw(bgTree4CNode_typ* node1, bgTree4CNode_typ* node2)
{
#ifdef WIN32
    if( node1->dw ){
        DBGMSG("bgTree4CNodeAddDw(): node1(id=%d) has dw(id=%d)\n ", node1->id, node1->dw->id);
    }

    if( node2->up ){
        DBGMSG("bgTree4CNodeAddDw(): node2(id=%d) has up(id=%d)\n ", node2->id, node2->up->id);
    }
#endif

    node1->dw = node2;
    node2->up = node1;
}

int bgTree4CNodeAppendToDwEnd(bgTree4CNode_typ* node1, bgTree4CNode_typ* node2)
{
bgTree4CNode_typ* n1 = node1;
bgTree4CNode_typ* n2;
int i;

    for(i=0;i<node1->nodeCountMax;i++){
        n2 = n1->dw;
        if( n2 )
            n1 = n2;
        else{
            n1->dw = node2;
			node2->up = n1;
            return 0;
        }
    }

    return 1;
}

void bgTree4CNodeAddRt(bgTree4CNode_typ* node1, bgTree4CNode_typ* node2)
{
#ifdef WIN32
    if( node1->rt ){
        DBGMSG("bgTree4CNodeAddDw(): node1(id=%d) has rt(id=%d)\n ", node1->id, node1->rt->id);
    }

    if( node2->lf ){
        DBGMSG("bgTree4CNodeAddDw(): node2(id=%d) has lf(id=%d)\n ", node2->id, node2->lf->id);
    }
#endif

    node1->rt = node2;
    node2->lf = node1;
}

int bgTree4CNodeAppendToRtEnd(bgTree4CNode_typ* node1, bgTree4CNode_typ* node2)
{
bgTree4CNode_typ* n1 = node1;
bgTree4CNode_typ* n2;
int i;

    for(i=0;i<node1->nodeCountMax;i++){
        n2 = n1->rt;
        if( n2 )
            n1 = n2;
        else{
            n1->rt = node2;
            return 0;
        }
    }

    return 1;
}

int	bgTree4CNodeInsertRt(bgTree4CNode_typ* node1, bgTree4CNode_typ* node2)
{
bgTree4CNode_typ* pNode;

	pNode = node1->rt;
	if( pNode ){
		pNode->lf = node2;
		node1->rt = node2;
		node2->lf = node1;
		node2->rt = pNode;
	}else{
		node1->rt = node2;
		node2->lf = node1;
	}
	return 0;
}

int	bgTree4CNodeInsertLf(bgTree4CNode_typ* node1, bgTree4CNode_typ* node2)
{
bgTree4CNode_typ* pNode;

	pNode = node1->lf;
	if( pNode ){
		pNode->rt = node2;
		node1->lf = node2;
		node2->rt = node1;
		node2->lf = pNode;
	}else{
		node1->lf = node2;
		node2->rt = node1;
	}
	return 0;
}

bgTree4CNode_typ* bgTree4CGetNextNodeRtDw(bgTree4CNode_typ* n1)
{
bgTree4CNode_typ* n2;

	if( !n1 )
		return 0;

	/*is node on the right of the current node defined?*/
	n2 = n1->rt;
    if( n2 ){
		/*right node found!*/
		return n2;
    }

	/*current node has no "right" nodes*/

	/*any down nodes from the current node?*/
    n2 = n1->dw;

    if( n2 ){
		/*down node found!*/
		return n2;
    }

	return 0;
}

bgTree4CNode_typ* bgTree4CGetNextNodeDw(bgTree4CNode_typ* n1)
{
	if( !n1 )
		return 0;

	/*any down nodes from the current node?*/
    return n1->dw;

}

void bgTree4CNodeSetDataType(bgTree4CNode_typ* node, int dataType)
{
    node->dataType = dataType;
}

void bgTree4CNodeSetDataValue(bgTree4CNode_typ* node, int dataVal)
{
    node->dataValue = dataVal;
}

void bgTree4CNodeSetDataPtr(bgTree4CNode_typ* node, char* data)
{
    node->data = data;
}

int bgTree4CNodeGetDataType(bgTree4CNode_typ* node)
{
    return node->dataType;
}

int bgTree4CNodeGetDataValue(bgTree4CNode_typ* node)
{
    return node->dataValue;
}

char* bgTree4CNodeGetDataPtr(bgTree4CNode_typ* node)
{
    return node->data;
}

void bgTree4CPrint(bgTree4C_typ* tree)
{
/*start w. root*/
bgTree4CNode_typ* n1 = &tree->nodes[0];
bgTree4CNode_typ* n2;
bgStack_typ stack;
bgStack_typ* s = &stack;

    bgStackInit(s);
    while(1){

		/*check if curent node exists*/
        if(!n1)
            return;

		/*display current node info*/
/*
        DBGMSG("%sid=%d, type=%s, data=%s\n", pTabs[bgStackGetItemCount(s)], n1->id, xmlRpcKeywDict[n1->dataType], n1->data?n1->data:"nil");
*/
#ifdef WIN32
		if(n1->data)
	        DBGMSG("nId=%d %s Type=%d [%s] Value=%d\n", n1->id, pTabs[bgStackGetItemCount(s)], n1->dataType, n1->data?n1->data:"?", n1->dataValue);
		else
	        DBGMSG("nId=%d %s Type=%d Value=%d\n", n1->id, pTabs[bgStackGetItemCount(s)], n1->dataType, n1->dataValue);
#endif

		/*first, print all nodes on the right from the current node*/

		/*is node on the right of the current node defined?*/
		n2 = n1->rt;
        if( n2 ){
			/*yes, right node defined; push current node to stack*/
            bgStackPush(s, (char*) n1);
			/*current node becomes the node from the right; noOfItemsOnTheStack == level is now increased!*/
			n1 = n2;
            continue;
        }

		/*current node has no more "right" nodes*/

		/*any down nodes from the current node?*/
        n2 = n1->dw;

        if( n2 ){
			/*down node found; new current node is that node*/
            n1 = n2;
            continue;
        }

		/*current node has no more rigth & no more down nodes;
		find a node from the stack that has a down node defined
		*/
		while(1){

			if(!bgStackGetItemCount(s))
				return;

			n2 = (bgTree4CNode_typ*)bgStackPop(s);

			if( n2 ){
				n1 = n2->dw;
				if( !n1 )
					continue;
				else
					break;
			}
		}

	}
}

#endif
```
